ABB RAPID module: etna.mod

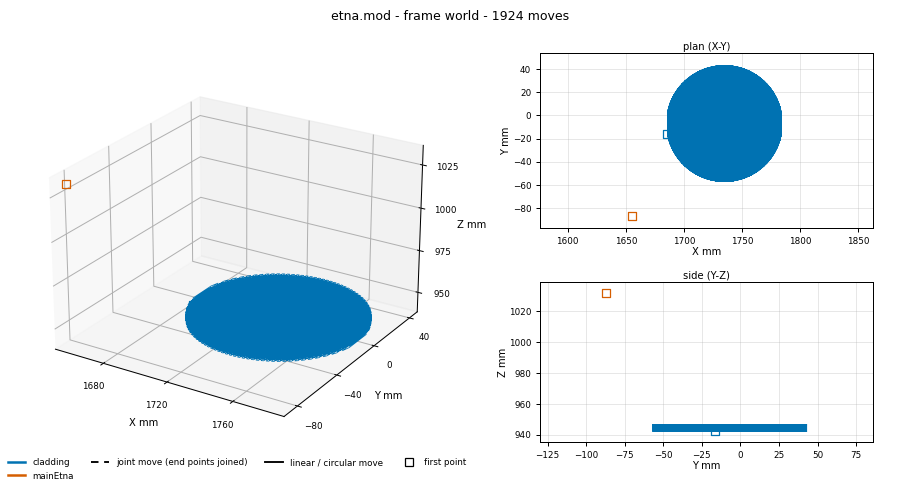
[picture p0: tool path of etna.mod in frame world, 1924 of 1924 moves have a stored position in this frame; points joined in program order, loops and branches not executed]
MODULE Etna

    PERS tooldata toolEtna:=[TRUE,[[530.0,46.8,126.6],[0.707107,0.000000,0.707107,0.000000]],[20,[70,30,123.5],[0,0,1,0],1,0,1]];
    PERS wobjdata wobjEtna:=[FALSE,TRUE,"",[[1655.0,-87.0,932.0],[1.000000,0.000000,0.000000,0.000000]],[[0,0,0],[1,0,0,0]]];

    VAR triggdata laserON;
    VAR triggdata laserOFF;

    CONST speeddata vl:=[10,500,5000,1000];


    CONST robtarget T0:=[[30.859828,70.797151,10.399975],[0.000000,0.000000,1.000000,0.000000],[0,0,-1,0],[9E+09,9E+09,9E+09,9E+09,9E+09,9E+09]];
    CONST robtarget T1:=[[30.859828,89.202857,10.399975],[0.000000,0.000000,1.000000,0.000000],[0,0,-1,0],[9E+09,9E+09,9E+09,9E+09,9E+09,9E+09]];
    CONST robtarget T2:=[[30.859828,70.797151,10.399975],[0.000000,0.000000,1.000000,0.000000],[0,0,-1,0],[9E+09,9E+09,9E+09,9E+09,9E+09,9E+09]];
    CONST robtarget T3:=[[30.859828,89.202857,10.399975],[0.000000,0.000000,1.000000,0.000000],[0,0,-1,0],[9E+09,9E+09,9E+09,9E+09,9E+09,9E+09]];
    CONST robtarget T4:=[[32.119833,94.360756,10.399975],[0.000000,0.000000,1.000000,0.000000],[0,0,-1,0],[9E+09,9E+09,9E+09,9E+09,9E+09,9E+09]];
    CONST robtarget T5:=[[32.119833,65.639251,10.399975],[0.000000,0.000000,1.000000,0.000000],[0,0,-1,0],[9E+09,9E+09,9E+09,9E+09,9E+09,9E+09]];
    CONST robtarget T6:=[[33.379837,61.953657,10.399975],[0.000000,0.000000,1.000000,0.000000],[0,0,-1,0],[9E+09,9E+09,9E+09,9E+09,9E+09,9E+09]];
    CONST robtarget T7:=[[33.379837,98.046351,10.399975],[0.000000,0.000000,1.000000,0.000000],[0,0,-1,0],[9E+09,9E+09,9E+09,9E+09,9E+09,9E+09]];
    CONST robtarget T8:=[[34.639842,101.007928,10.399975],[0.000000,0.000000,1.000000,0.000000],[0,0,-1,0],[9E+09,9E+09,9E+09,9E+09,9E+09,9E+09]];
    CONST robtarget T9:=[[34.639842,58.992080,10.399975],[0.000000,0.000000,1.000000,0.000000],[0,0,-1,0],[9E+09,9E+09,9E+09,9E+09,9E+09,9E+09]];
    CONST robtarget T10:=[[35.899846,56.444690,10.399975],[0.000000,0.000000,1.000000,0.000000],[0,0,-1,0],[9E+09,9E+09,9E+09,9E+09,9E+09,9E+09]];
    CONST robtarget T11:=[[35.899846,103.555317,10.399975],[0.000000,0.000000,1.000000,0.000000],[0,0,-1,0],[9E+09,9E+09,9E+09,9E+09,9E+09,9E+09]];
    CONST robtarget T12:=[[37.159851,105.775934,10.399975],[0.000000,0.000000,1.000000,0.000000],[0,0,-1,0],[9E+09,9E+09,9E+09,9E+09,9E+09,9E+09]];
    CONST robtarget T13:=[[37.159851,54.224074,10.399975],[0.000000,0.000000,1.000000,0.000000],[0,0,-1,0],[9E+09,9E+09,9E+09,9E+09,9E+09,9E+09]];
    CONST robtarget T14:=[[38.419855,52.240778,10.399975],[0.000000,0.000000,1.000000,0.000000],[0,0,-1,0],[9E+09,9E+09,9E+09,9E+09,9E+09,9E+09]];
    CONST robtarget T15:=[[38.419855,76.422528,10.399975],[0.000000,0.000000,1.000000,0.000000],[0,0,-1,0],[9E+09,9E+09,9E+09,9E+09,9E+09,9E+09]];
    CONST robtarget T16:=[[38.419855,83.577479,10.399975],[0.000000,0.000000,1.000000,0.000000],[0,0,-1,0],[9E+09,9E+09,9E+09,9E+09,9E+09,9E+09]];
    CONST robtarget T17:=[[38.419855,107.759230,10.399975],[0.000000,0.000000,1.000000,0.000000],[0,0,-1,0],[9E+09,9E+09,9E+09,9E+09,9E+09,9E+09]];
    CONST robtarget T18:=[[39.679860,109.560940,10.399975],[0.000000,0.000000,1.000000,0.000000],[0,0,-1,0],[9E+09,9E+09,9E+09,9E+09,9E+09,9E+09]];
    CONST robtarget T19:=[[39.679860,85.271589,10.399975],[0.000000,0.000000,1.000000,0.000000],[0,0,-1,0],[9E+09,9E+09,9E+09,9E+09,9E+09,9E+09]];
    CONST robtarget T20:=[[39.679860,74.728418,10.399975],[0.000000,0.000000,1.000000,0.000000],[0,0,-1,0],[9E+09,9E+09,9E+09,9E+09,9E+09,9E+09]];
    CONST robtarget T21:=[[39.679860,50.439068,10.399975],[0.000000,0.000000,1.000000,0.000000],[0,0,-1,0],[9E+09,9E+09,9E+09,9E+09,9E+09,9E+09]];
    CONST robtarget T22:=[[40.939864,48.787854,10.399975],[0.000000,0.000000,1.000000,0.000000],[0,0,-1,0],[9E+09,9E+09,9E+09,9E+09,9E+09,9E+09]];
    CONST robtarget T23:=[[40.939864,73.708792,10.399975],[0.000000,0.000000,1.000000,0.000000],[0,0,-1,0],[9E+09,9E+09,9E+09,9E+09,9E+09,9E+09]];
    CONST robtarget T24:=[[40.939864,86.291215,10.399975],[0.000000,0.000000,1.000000,0.000000],[0,0,-1,0],[9E+09,9E+09,9E+09,9E+09,9E+09,9E+09]];
    CONST robtarget T25:=[[40.939864,111.212154,10.399975],[0.000000,0.000000,1.000000,0.000000],[0,0,-1,0],[9E+09,9E+09,9E+09,9E+09,9E+09,9E+09]];
    CONST robtarget T26:=[[42.199869,112.721391,10.399975],[0.000000,0.000000,1.000000,0.000000],[0,0,-1,0],[9E+09,9E+09,9E+09,9E+09,9E+09,9E+09]];
    CONST robtarget T27:=[[42.199869,86.948670,10.399975],[0.000000,0.000000,1.000000,0.000000],[0,0,-1,0],[9E+09,9E+09,9E+09,9E+09,9E+09,9E+09]];
    CONST robtarget T28:=[[42.199869,73.051337,10.399975],[0.000000,0.000000,1.000000,0.000000],[0,0,-1,0],[9E+09,9E+09,9E+09,9E+09,9E+09,9E+09]];
    CONST robtarget T29:=[[42.199869,47.278617,10.399975],[0.000000,0.000000,1.000000,0.000000],[0,0,-1,0],[9E+09,9E+09,9E+09,9E+09,9E+09,9E+09]];
    CONST robtarget T30:=[[43.459873,45.884908,10.399975],[0.000000,0.000000,1.000000,0.000000],[0,0,-1,0],[9E+09,9E+09,9E+09,9E+09,9E+09,9E+09]];
    CONST robtarget T31:=[[43.459873,72.670297,10.399975],[0.000000,0.000000,1.000000,0.000000],[0,0,-1,0],[9E+09,9E+09,9E+09,9E+09,9E+09,9E+09]];
    CONST robtarget T32:=[[43.459873,87.329711,10.399975],[0.000000,0.000000,1.000000,0.000000],[0,0,-1,0],[9E+09,9E+09,9E+09,9E+09,9E+09,9E+09]];
    CONST robtarget T33:=[[43.459873,114.115099,10.399975],[0.000000,0.000000,1.000000,0.000000],[0,0,-1,0],[9E+09,9E+09,9E+09,9E+09,9E+09,9E+09]];
    CONST robtarget T34:=[[44.719878,115.412758,10.399975],[0.000000,0.000000,1.000000,0.000000],[0,0,-1,0],[9E+09,9E+09,9E+09,9E+09,9E+09,9E+09]];
    CONST robtarget T35:=[[44.719878,87.487316,10.399975],[0.000000,0.000000,1.000000,0.000000],[0,0,-1,0],[9E+09,9E+09,9E+09,9E+09,9E+09,9E+09]];
    CONST robtarget T36:=[[44.719878,72.512692,10.399975],[0.000000,0.000000,1.000000,0.000000],[0,0,-1,0],[9E+09,9E+09,9E+09,9E+09,9E+09,9E+09]];
    CONST robtarget T37:=[[44.719878,44.587250,10.399975],[0.000000,0.000000,1.000000,0.000000],[0,0,-1,0],[9E+09,9E+09,9E+09,9E+09,9E+09,9E+09]];
    CONST robtarget T38:=[[45.979882,43.373063,10.399975],[0.000000,0.000000,1.000000,0.000000],[0,0,-1,0],[9E+09,9E+09,9E+09,9E+09,9E+09,9E+09]];
    CONST robtarget T39:=[[45.979882,72.576253,10.399975],[0.000000,0.000000,1.000000,0.000000],[0,0,-1,0],[9E+09,9E+09,9E+09,9E+09,9E+09,9E+09]];
    CONST robtarget T40:=[[45.979882,87.423755,10.399975],[0.000000,0.000000,1.000000,0.000000],[0,0,-1,0],[9E+09,9E+09,9E+09,9E+09,9E+09,9E+09]];
    CONST robtarget T41:=[[45.979882,116.626944,10.399975],[0.000000,0.000000,1.000000,0.000000],[0,0,-1,0],[9E+09,9E+09,9E+09,9E+09,9E+09,9E+09]];
    CONST robtarget T42:=[[47.239887,117.767805,10.399975],[0.000000,0.000000,1.000000,0.000000],[0,0,-1,0],[9E+09,9E+09,9E+09,9E+09,9E+09,9E+09]];
    CONST robtarget T43:=[[47.239887,87.152583,10.399975],[0.000000,0.000000,1.000000,0.000000],[0,0,-1,0],[9E+09,9E+09,9E+09,9E+09,9E+09,9E+09]];
    CONST robtarget T44:=[[47.239887,72.847425,10.399975],[0.000000,0.000000,1.000000,0.000000],[0,0,-1,0],[9E+09,9E+09,9E+09,9E+09,9E+09,9E+09]];
    CONST robtarget T45:=[[47.239887,42.232203,10.399975],[0.000000,0.000000,1.000000,0.000000],[0,0,-1,0],[9E+09,9E+09,9E+09,9E+09,9E+09,9E+09]];
    CONST robtarget T46:=[[48.499891,41.180273,10.399975],[0.000000,0.000000,1.000000,0.000000],[0,0,-1,0],[9E+09,9E+09,9E+09,9E+09,9E+09,9E+09]];
    CONST robtarget T47:=[[48.499891,73.379202,10.399975],[0.000000,0.000000,1.000000,0.000000],[0,0,-1,0],[9E+09,9E+09,9E+09,9E+09,9E+09,9E+09]];
    CONST robtarget T48:=[[48.499891,86.620805,10.399975],[0.000000,0.000000,1.000000,0.000000],[0,0,-1,0],[9E+09,9E+09,9E+09,9E+09,9E+09,9E+09]];
    CONST robtarget T49:=[[48.499891,118.819735,10.399975],[0.000000,0.000000,1.000000,0.000000],[0,0,-1,0],[9E+09,9E+09,9E+09,9E+09,9E+09,9E+09]];
    CONST robtarget T50:=[[49.759896,119.803025,10.399975],[0.000000,0.000000,1.000000,0.000000],[0,0,-1,0],[9E+09,9E+09,9E+09,9E+09,9E+09,9E+09]];
    CONST robtarget T51:=[[49.759896,85.779969,10.399975],[0.000000,0.000000,1.000000,0.000000],[0,0,-1,0],[9E+09,9E+09,9E+09,9E+09,9E+09,9E+09]];
    CONST robtarget T52:=[[49.759896,74.220038,10.399975],[0.000000,0.000000,1.000000,0.000000],[0,0,-1,0],[9E+09,9E+09,9E+09,9E+09,9E+09,9E+09]];
    CONST robtarget T53:=[[49.759896,40.196983,10.399975],[0.000000,0.000000,1.000000,0.000000],[0,0,-1,0],[9E+09,9E+09,9E+09,9E+09,9E+09,9E+09]];
    CONST robtarget T54:=[[51.019900,39.265681,10.399975],[0.000000,0.000000,1.000000,0.000000],[0,0,-1,0],[9E+09,9E+09,9E+09,9E+09,9E+09,9E+09]];
    CONST robtarget T55:=[[51.019900,75.547902,10.399975],[0.000000,0.000000,1.000000,0.000000],[0,0,-1,0],[9E+09,9E+09,9E+09,9E+09,9E+09,9E+09]];
    CONST robtarget T56:=[[51.019900,84.452106,10.399975],[0.000000,0.000000,1.000000,0.000000],[0,0,-1,0],[9E+09,9E+09,9E+09,9E+09,9E+09,9E+09]];
    CONST robtarget T57:=[[51.019900,120.734326,10.399975],[0.000000,0.000000,1.000000,0.000000],[0,0,-1,0],[9E+09,9E+09,9E+09,9E+09,9E+09,9E+09]];
    CONST robtarget T58:=[[52.279905,121.607260,10.399975],[0.000000,0.000000,1.000000,0.000000],[0,0,-1,0],[9E+09,9E+09,9E+09,9E+09,9E+09,9E+09]];
    CONST robtarget T59:=[[52.279905,81.789524,10.399975],[0.000000,0.000000,1.000000,0.000000],[0,0,-1,0],[9E+09,9E+09,9E+09,9E+09,9E+09,9E+09]];
    CONST robtarget T60:=[[52.279905,78.210483,10.399975],[0.000000,0.000000,1.000000,0.000000],[0,0,-1,0],[9E+09,9E+09,9E+09,9E+09,9E+09,9E+09]];
    CONST robtarget T61:=[[52.279905,38.392748,10.399975],[0.000000,0.000000,1.000000,0.000000],[0,0,-1,0],[9E+09,9E+09,9E+09,9E+09,9E+09,9E+09]];
    CONST robtarget T62:=[[53.539909,37.589739,10.399975],[0.000000,0.000000,1.000000,0.000000],[0,0,-1,0],[9E+09,9E+09,9E+09,9E+09,9E+09,9E+09]];
    CONST robtarget T63:=[[53.539909,122.410268,10.399975],[0.000000,0.000000,1.000000,0.000000],[0,0,-1,0],[9E+09,9E+09,9E+09,9E+09,9E+09,9E+09]];
    CONST robtarget T64:=[[54.799914,123.174878,10.399975],[0.000000,0.000000,1.000000,0.000000],[0,0,-1,0],[9E+09,9E+09,9E+09,9E+09,9E+09,9E+09]];
    CONST robtarget T65:=[[54.799914,36.825129,10.399975],[0.000000,0.000000,1.000000,0.000000],[0,0,-1,0],[9E+09,9E+09,9E+09,9E+09,9E+09,9E+09]];
    CONST robtarget T66:=[[56.059918,36.110177,10.399975],[0.000000,0.000000,1.000000,0.000000],[0,0,-1,0],[9E+09,9E+09,9E+09,9E+09,9E+09,9E+09]];
    CONST robtarget T67:=[[56.059918,123.889831,10.399975],[0.000000,0.000000,1.000000,0.000000],[0,0,-1,0],[9E+09,9E+09,9E+09,9E+09,9E+09,9E+09]];
    CONST robtarget T68:=[[57.319923,124.546114,10.399975],[0.000000,0.000000,1.000000,0.000000],[0,0,-1,0],[9E+09,9E+09,9E+09,9E+09,9E+09,9E+09]];
    CONST robtarget T69:=[[57.319923,35.453894,10.399975],[0.000000,0.000000,1.000000,0.000000],[0,0,-1,0],[9E+09,9E+09,9E+09,9E+09,9E+09,9E+09]];
    CONST robtarget T70:=[[58.579927,34.827050,10.399975],[0.000000,0.000000,1.000000,0.000000],[0,0,-1,0],[9E+09,9E+09,9E+09,9E+09,9E+09,9E+09]];
    CONST robtarget T71:=[[58.579927,125.172958,10.399975],[0.000000,0.000000,1.000000,0.000000],[0,0,-1,0],[9E+09,9E+09,9E+09,9E+09,9E+09,9E+09]];
    CONST robtarget T72:=[[59.839932,125.745278,10.399975],[0.000000,0.000000,1.000000,0.000000],[0,0,-1,0],[9E+09,9E+09,9E+09,9E+09,9E+09,9E+09]];
    CONST robtarget T73:=[[59.839932,34.254730,10.399975],[0.000000,0.000000,1.000000,0.000000],[0,0,-1,0],[9E+09,9E+09,9E+09,9E+09,9E+09,9E+09]];
    CONST robtarget T74:=[[61.099936,33.722290,10.399975],[0.000000,0.000000,1.000000,0.000000],[0,0,-1,0],[9E+09,9E+09,9E+09,9E+09,9E+09,9E+09]];
    CONST robtarget T75:=[[61.099936,126.277717,10.399975],[0.000000,0.000000,1.000000,0.000000],[0,0,-1,0],[9E+09,9E+09,9E+09,9E+09,9E+09,9E+09]];
    CONST robtarget T76:=[[62.359941,126.783143,10.399975],[0.000000,0.000000,1.000000,0.000000],[0,0,-1,0],[9E+09,9E+09,9E+09,9E+09,9E+09,9E+09]];
    CONST robtarget T77:=[[62.359941,33.216864,10.399975],[0.000000,0.000000,1.000000,0.000000],[0,0,-1,0],[9E+09,9E+09,9E+09,9E+09,9E+09,9E+09]];
    CONST robtarget T78:=[[63.619945,32.772318,10.399975],[0.000000,0.000000,1.000000,0.000000],[0,0,-1,0],[9E+09,9E+09,9E+09,9E+09,9E+09,9E+09]];
    CONST robtarget T79:=[[63.619945,127.227690,10.399975],[0.000000,0.000000,1.000000,0.000000],[0,0,-1,0],[9E+09,9E+09,9E+09,9E+09,9E+09,9E+09]];
    CONST robtarget T80:=[[64.879950,127.652167,10.399975],[0.000000,0.000000,1.000000,0.000000],[0,0,-1,0],[9E+09,9E+09,9E+09,9E+09,9E+09,9E+09]];
    CONST robtarget T81:=[[64.879950,32.347841,10.399975],[0.000000,0.000000,1.000000,0.000000],[0,0,-1,0],[9E+09,9E+09,9E+09,9E+09,9E+09,9E+09]];
    CONST robtarget T82:=[[66.139954,31.969479,10.399975],[0.000000,0.000000,1.000000,0.000000],[0,0,-1,0],[9E+09,9E+09,9E+09,9E+09,9E+09,9E+09]];
    CONST robtarget T83:=[[66.139954,128.030529,10.399975],[0.000000,0.000000,1.000000,0.000000],[0,0,-1,0],[9E+09,9E+09,9E+09,9E+09,9E+09,9E+09]];
    CONST robtarget T84:=[[67.399959,128.374988,10.399975],[0.000000,0.000000,1.000000,0.000000],[0,0,-1,0],[9E+09,9E+09,9E+09,9E+09,9E+09,9E+09]];
    CONST robtarget T85:=[[67.399959,31.625019,10.399975],[0.000000,0.000000,1.000000,0.000000],[0,0,-1,0],[9E+09,9E+09,9E+09,9E+09,9E+09,9E+09]];
    CONST robtarget T86:=[[68.659963,31.307526,10.399975],[0.000000,0.000000,1.000000,0.000000],[0,0,-1,0],[9E+09,9E+09,9E+09,9E+09,9E+09,9E+09]];
    CONST robtarget T87:=[[68.659963,128.692481,10.399975],[0.000000,0.000000,1.000000,0.000000],[0,0,-1,0],[9E+09,9E+09,9E+09,9E+09,9E+09,9E+09]];
    CONST robtarget T88:=[[69.919968,128.960575,10.399975],[0.000000,0.000000,1.000000,0.000000],[0,0,-1,0],[9E+09,9E+09,9E+09,9E+09,9E+09,9E+09]];
    CONST robtarget T89:=[[69.919968,31.039433,10.399975],[0.000000,0.000000,1.000000,0.000000],[0,0,-1,0],[9E+09,9E+09,9E+09,9E+09,9E+09,9E+09]];
    CONST robtarget T90:=[[71.179972,30.786444,10.399975],[0.000000,0.000000,1.000000,0.000000],[0,0,-1,0],[9E+09,9E+09,9E+09,9E+09,9E+09,9E+09]];
    CONST robtarget T91:=[[71.179972,129.213563,10.399975],[0.000000,0.000000,1.000000,0.000000],[0,0,-1,0],[9E+09,9E+09,9E+09,9E+09,9E+09,9E+09]];
    CONST robtarget T92:=[[72.439977,129.413129,10.399975],[0.000000,0.000000,1.000000,0.000000],[0,0,-1,0],[9E+09,9E+09,9E+09,9E+09,9E+09,9E+09]];
    CONST robtarget T93:=[[72.439977,30.586879,10.399975],[0.000000,0.000000,1.000000,0.000000],[0,0,-1,0],[9E+09,9E+09,9E+09,9E+09,9E+09,9E+09]];
    CONST robtarget T94:=[[73.699981,30.406130,10.399975],[0.000000,0.000000,1.000000,0.000000],[0,0,-1,0],[9E+09,9E+09,9E+09,9E+09,9E+09,9E+09]];
    CONST robtarget T95:=[[73.699981,40.937335,10.399975],[0.000000,0.000000,1.000000,0.000000],[0,0,-1,0],[9E+09,9E+09,9E+09,9E+09,9E+09,9E+09]];
    CONST robtarget T96:=[[73.699981,49.062665,10.399975],[0.000000,0.000000,1.000000,0.000000],[0,0,-1,0],[9E+09,9E+09,9E+09,9E+09,9E+09,9E+09]];
    CONST robtarget T97:=[[73.699981,75.937339,10.399975],[0.000000,0.000000,1.000000,0.000000],[0,0,-1,0],[9E+09,9E+09,9E+09,9E+09,9E+09,9E+09]];
    CONST robtarget T98:=[[73.699981,84.062668,10.399975],[0.000000,0.000000,1.000000,0.000000],[0,0,-1,0],[9E+09,9E+09,9E+09,9E+09,9E+09,9E+09]];
    CONST robtarget T99:=[[73.699981,110.937342,10.399975],[0.000000,0.000000,1.000000,0.000000],[0,0,-1,0],[9E+09,9E+09,9E+09,9E+09,9E+09,9E+09]];
    CONST robtarget T100:=[[73.699981,119.062672,10.399975],[0.000000,0.000000,1.000000,0.000000],[0,0,-1,0],[9E+09,9E+09,9E+09,9E+09,9E+09,9E+09]];
    CONST robtarget T101:=[[73.699981,129.593877,10.399975],[0.000000,0.000000,1.000000,0.000000],[0,0,-1,0],[9E+09,9E+09,9E+09,9E+09,9E+09,9E+09]];
    CONST robtarget T102:=[[74.959986,129.735844,10.399975],[0.000000,0.000000,1.000000,0.000000],[0,0,-1,0],[9E+09,9E+09,9E+09,9E+09,9E+09,9E+09]];
    CONST robtarget T103:=[[74.959986,120.544921,10.399975],[0.000000,0.000000,1.000000,0.000000],[0,0,-1,0],[9E+09,9E+09,9E+09,9E+09,9E+09,9E+09]];
    CONST robtarget T104:=[[74.959986,109.455091,10.399975],[0.000000,0.000000,1.000000,0.000000],[0,0,-1,0],[9E+09,9E+09,9E+09,9E+09,9E+09,9E+09]];
    CONST robtarget T105:=[[74.959986,85.544918,10.399975],[0.000000,0.000000,1.000000,0.000000],[0,0,-1,0],[9E+09,9E+09,9E+09,9E+09,9E+09,9E+09]];
    CONST robtarget T106:=[[74.959986,74.455090,10.399975],[0.000000,0.000000,1.000000,0.000000],[0,0,-1,0],[9E+09,9E+09,9E+09,9E+09,9E+09,9E+09]];
    CONST robtarget T107:=[[74.959986,50.544916,10.399975],[0.000000,0.000000,1.000000,0.000000],[0,0,-1,0],[9E+09,9E+09,9E+09,9E+09,9E+09,9E+09]];
    CONST robtarget T108:=[[74.959986,39.455086,10.399975],[0.000000,0.000000,1.000000,0.000000],[0,0,-1,0],[9E+09,9E+09,9E+09,9E+09,9E+09,9E+09]];
    CONST robtarget T109:=[[74.959986,30.264163,10.399975],[0.000000,0.000000,1.000000,0.000000],[0,0,-1,0],[9E+09,9E+09,9E+09,9E+09,9E+09,9E+09]];
    CONST robtarget T110:=[[76.219990,30.153959,10.399975],[0.000000,0.000000,1.000000,0.000000],[0,0,-1,0],[9E+09,9E+09,9E+09,9E+09,9E+09,9E+09]];
    CONST robtarget T111:=[[76.219990,38.524551,10.399975],[0.000000,0.000000,1.000000,0.000000],[0,0,-1,0],[9E+09,9E+09,9E+09,9E+09,9E+09,9E+09]];
    CONST robtarget T112:=[[76.219990,51.475451,10.399975],[0.000000,0.000000,1.000000,0.000000],[0,0,-1,0],[9E+09,9E+09,9E+09,9E+09,9E+09,9E+09]];
    CONST robtarget T113:=[[76.219990,73.524553,10.399975],[0.000000,0.000000,1.000000,0.000000],[0,0,-1,0],[9E+09,9E+09,9E+09,9E+09,9E+09,9E+09]];
    CONST robtarget T114:=[[76.219990,86.475455,10.399975],[0.000000,0.000000,1.000000,0.000000],[0,0,-1,0],[9E+09,9E+09,9E+09,9E+09,9E+09,9E+09]];
    CONST robtarget T115:=[[76.219990,108.524556,10.399975],[0.000000,0.000000,1.000000,0.000000],[0,0,-1,0],[9E+09,9E+09,9E+09,9E+09,9E+09,9E+09]];
    CONST robtarget T116:=[[76.219990,121.475457,10.399975],[0.000000,0.000000,1.000000,0.000000],[0,0,-1,0],[9E+09,9E+09,9E+09,9E+09,9E+09,9E+09]];
    CONST robtarget T117:=[[76.219990,129.846049,10.399975],[0.000000,0.000000,1.000000,0.000000],[0,0,-1,0],[9E+09,9E+09,9E+09,9E+09,9E+09,9E+09]];
    CONST robtarget T118:=[[77.479995,129.931001,10.399975],[0.000000,0.000000,1.000000,0.000000],[0,0,-1,0],[9E+09,9E+09,9E+09,9E+09,9E+09,9E+09]];
    CONST robtarget T119:=[[77.479995,122.050628,10.399975],[0.000000,0.000000,1.000000,0.000000],[0,0,-1,0],[9E+09,9E+09,9E+09,9E+09,9E+09,9E+09]];
    CONST robtarget T120:=[[77.479995,107.949384,10.399975],[0.000000,0.000000,1.000000,0.000000],[0,0,-1,0],[9E+09,9E+09,9E+09,9E+09,9E+09,9E+09]];
    CONST robtarget T121:=[[77.479995,87.050626,10.399975],[0.000000,0.000000,1.000000,0.000000],[0,0,-1,0],[9E+09,9E+09,9E+09,9E+09,9E+09,9E+09]];
    CONST robtarget T122:=[[77.479995,72.949381,10.399975],[0.000000,0.000000,1.000000,0.000000],[0,0,-1,0],[9E+09,9E+09,9E+09,9E+09,9E+09,9E+09]];
    CONST robtarget T123:=[[77.479995,52.050624,10.399975],[0.000000,0.000000,1.000000,0.000000],[0,0,-1,0],[9E+09,9E+09,9E+09,9E+09,9E+09,9E+09]];
    CONST robtarget T124:=[[77.479995,37.949379,10.399975],[0.000000,0.000000,1.000000,0.000000],[0,0,-1,0],[9E+09,9E+09,9E+09,9E+09,9E+09,9E+09]];
    CONST robtarget T125:=[[77.479995,30.069007,10.399975],[0.000000,0.000000,1.000000,0.000000],[0,0,-1,0],[9E+09,9E+09,9E+09,9E+09,9E+09,9E+09]];
    CONST robtarget T126:=[[78.739999,30.028279,10.399975],[0.000000,0.000000,1.000000,0.000000],[0,0,-1,0],[9E+09,9E+09,9E+09,9E+09,9E+09,9E+09]];
    CONST robtarget T127:=[[78.739999,37.608991,10.399975],[0.000000,0.000000,1.000000,0.000000],[0,0,-1,0],[9E+09,9E+09,9E+09,9E+09,9E+09,9E+09]];
    CONST robtarget T128:=[[78.739999,52.391011,10.399975],[0.000000,0.000000,1.000000,0.000000],[0,0,-1,0],[9E+09,9E+09,9E+09,9E+09,9E+09,9E+09]];
    CONST robtarget T129:=[[78.739999,72.608994,10.399975],[0.000000,0.000000,1.000000,0.000000],[0,0,-1,0],[9E+09,9E+09,9E+09,9E+09,9E+09,9E+09]];
    CONST robtarget T130:=[[78.739999,87.391014,10.399975],[0.000000,0.000000,1.000000,0.000000],[0,0,-1,0],[9E+09,9E+09,9E+09,9E+09,9E+09,9E+09]];
    CONST robtarget T131:=[[78.739999,107.608996,10.399975],[0.000000,0.000000,1.000000,0.000000],[0,0,-1,0],[9E+09,9E+09,9E+09,9E+09,9E+09,9E+09]];
    CONST robtarget T132:=[[78.739999,122.391017,10.399975],[0.000000,0.000000,1.000000,0.000000],[0,0,-1,0],[9E+09,9E+09,9E+09,9E+09,9E+09,9E+09]];
    CONST robtarget T133:=[[78.739999,129.971729,10.399975],[0.000000,0.000000,1.000000,0.000000],[0,0,-1,0],[9E+09,9E+09,9E+09,9E+09,9E+09,9E+09]];
    CONST robtarget T134:=[[80.000004,130.000008,10.399975],[0.000000,0.000000,1.000000,0.000000],[0,0,-1,0],[9E+09,9E+09,9E+09,9E+09,9E+09,9E+09]];
    CONST robtarget T135:=[[80.000004,122.487319,10.399975],[0.000000,0.000000,1.000000,0.000000],[0,0,-1,0],[9E+09,9E+09,9E+09,9E+09,9E+09,9E+09]];
    CONST robtarget T136:=[[80.000004,107.512696,10.399975],[0.000000,0.000000,1.000000,0.000000],[0,0,-1,0],[9E+09,9E+09,9E+09,9E+09,9E+09,9E+09]];
    CONST robtarget T137:=[[80.000004,87.487316,10.399975],[0.000000,0.000000,1.000000,0.000000],[0,0,-1,0],[9E+09,9E+09,9E+09,9E+09,9E+09,9E+09]];
    CONST robtarget T138:=[[80.000004,72.512692,10.399975],[0.000000,0.000000,1.000000,0.000000],[0,0,-1,0],[9E+09,9E+09,9E+09,9E+09,9E+09,9E+09]];
    CONST robtarget T139:=[[80.000004,52.487312,10.399975],[0.000000,0.000000,1.000000,0.000000],[0,0,-1,0],[9E+09,9E+09,9E+09,9E+09,9E+09,9E+09]];
    CONST robtarget T140:=[[80.000004,37.512688,10.399975],[0.000000,0.000000,1.000000,0.000000],[0,0,-1,0],[9E+09,9E+09,9E+09,9E+09,9E+09,9E+09]];
    CONST robtarget T141:=[[80.000004,30.000000,10.399975],[0.000000,0.000000,1.000000,0.000000],[0,0,-1,0],[9E+09,9E+09,9E+09,9E+09,9E+09,9E+09]];
    CONST robtarget T142:=[[81.260008,30.028279,10.399975],[0.000000,0.000000,1.000000,0.000000],[0,0,-1,0],[9E+09,9E+09,9E+09,9E+09,9E+09,9E+09]];
    CONST robtarget T143:=[[81.260008,37.608991,10.399975],[0.000000,0.000000,1.000000,0.000000],[0,0,-1,0],[9E+09,9E+09,9E+09,9E+09,9E+09,9E+09]];
    CONST robtarget T144:=[[81.260008,52.391011,10.399975],[0.000000,0.000000,1.000000,0.000000],[0,0,-1,0],[9E+09,9E+09,9E+09,9E+09,9E+09,9E+09]];
    CONST robtarget T145:=[[81.260008,72.608994,10.399975],[0.000000,0.000000,1.000000,0.000000],[0,0,-1,0],[9E+09,9E+09,9E+09,9E+09,9E+09,9E+09]];
    CONST robtarget T146:=[[81.260008,87.391014,10.399975],[0.000000,0.000000,1.000000,0.000000],[0,0,-1,0],[9E+09,9E+09,9E+09,9E+09,9E+09,9E+09]];
    CONST robtarget T147:=[[81.260008,107.608996,10.399975],[0.000000,0.000000,1.000000,0.000000],[0,0,-1,0],[9E+09,9E+09,9E+09,9E+09,9E+09,9E+09]];
    CONST robtarget T148:=[[81.260008,122.391017,10.399975],[0.000000,0.000000,1.000000,0.000000],[0,0,-1,0],[9E+09,9E+09,9E+09,9E+09,9E+09,9E+09]];
    CONST robtarget T149:=[[81.260008,129.971729,10.399975],[0.000000,0.000000,1.000000,0.000000],[0,0,-1,0],[9E+09,9E+09,9E+09,9E+09,9E+09,9E+09]];
    CONST robtarget T150:=[[82.520013,129.931001,10.399975],[0.000000,0.000000,1.000000,0.000000],[0,0,-1,0],[9E+09,9E+09,9E+09,9E+09,9E+09,9E+09]];
    CONST robtarget T151:=[[82.520013,122.050628,10.399975],[0.000000,0.000000,1.000000,0.000000],[0,0,-1,0],[9E+09,9E+09,9E+09,9E+09,9E+09,9E+09]];
    CONST robtarget T152:=[[82.520013,107.949384,10.399975],[0.000000,0.000000,1.000000,0.000000],[0,0,-1,0],[9E+09,9E+09,9E+09,9E+09,9E+09,9E+09]];
    CONST robtarget T153:=[[82.520013,87.050626,10.399975],[0.000000,0.000000,1.000000,0.000000],[0,0,-1,0],[9E+09,9E+09,9E+09,9E+09,9E+09,9E+09]];
    CONST robtarget T154:=[[82.520013,72.949381,10.399975],[0.000000,0.000000,1.000000,0.000000],[0,0,-1,0],[9E+09,9E+09,9E+09,9E+09,9E+09,9E+09]];
    CONST robtarget T155:=[[82.520013,52.050624,10.399975],[0.000000,0.000000,1.000000,0.000000],[0,0,-1,0],[9E+09,9E+09,9E+09,9E+09,9E+09,9E+09]];
    CONST robtarget T156:=[[82.520013,37.949379,10.399975],[0.000000,0.000000,1.000000,0.000000],[0,0,-1,0],[9E+09,9E+09,9E+09,9E+09,9E+09,9E+09]];
    CONST robtarget T157:=[[82.520013,30.069007,10.399975],[0.000000,0.000000,1.000000,0.000000],[0,0,-1,0],[9E+09,9E+09,9E+09,9E+09,9E+09,9E+09]];
    CONST robtarget T158:=[[83.780017,30.153959,10.399975],[0.000000,0.000000,1.000000,0.000000],[0,0,-1,0],[9E+09,9E+09,9E+09,9E+09,9E+09,9E+09]];
    CONST robtarget T159:=[[83.780017,38.524551,10.399975],[0.000000,0.000000,1.000000,0.000000],[0,0,-1,0],[9E+09,9E+09,9E+09,9E+09,9E+09,9E+09]];
    CONST robtarget T160:=[[83.780017,51.475451,10.399975],[0.000000,0.000000,1.000000,0.000000],[0,0,-1,0],[9E+09,9E+09,9E+09,9E+09,9E+09,9E+09]];
    CONST robtarget T161:=[[83.780017,73.524553,10.399975],[0.000000,0.000000,1.000000,0.000000],[0,0,-1,0],[9E+09,9E+09,9E+09,9E+09,9E+09,9E+09]];
    CONST robtarget T162:=[[83.780017,86.475455,10.399975],[0.000000,0.000000,1.000000,0.000000],[0,0,-1,0],[9E+09,9E+09,9E+09,9E+09,9E+09,9E+09]];
    CONST robtarget T163:=[[83.780017,108.524556,10.399975],[0.000000,0.000000,1.000000,0.000000],[0,0,-1,0],[9E+09,9E+09,9E+09,9E+09,9E+09,9E+09]];
    CONST robtarget T164:=[[83.780017,121.475457,10.399975],[0.000000,0.000000,1.000000,0.000000],[0,0,-1,0],[9E+09,9E+09,9E+09,9E+09,9E+09,9E+09]];
    CONST robtarget T165:=[[83.780017,129.846049,10.399975],[0.000000,0.000000,1.000000,0.000000],[0,0,-1,0],[9E+09,9E+09,9E+09,9E+09,9E+09,9E+09]];
    CONST robtarget T166:=[[85.040022,129.735844,10.399975],[0.000000,0.000000,1.000000,0.000000],[0,0,-1,0],[9E+09,9E+09,9E+09,9E+09,9E+09,9E+09]];
    CONST robtarget T167:=[[85.040022,120.544921,10.399975],[0.000000,0.000000,1.000000,0.000000],[0,0,-1,0],[9E+09,9E+09,9E+09,9E+09,9E+09,9E+09]];
    CONST robtarget T168:=[[85.040022,109.455091,10.399975],[0.000000,0.000000,1.000000,0.000000],[0,0,-1,0],[9E+09,9E+09,9E+09,9E+09,9E+09,9E+09]];
    CONST robtarget T169:=[[85.040022,85.544918,10.399975],[0.000000,0.000000,1.000000,0.000000],[0,0,-1,0],[9E+09,9E+09,9E+09,9E+09,9E+09,9E+09]];
    CONST robtarget T170:=[[85.040022,74.455090,10.399975],[0.000000,0.000000,1.000000,0.000000],[0,0,-1,0],[9E+09,9E+09,9E+09,9E+09,9E+09,9E+09]];
    CONST robtarget T171:=[[85.040022,50.544916,10.399975],[0.000000,0.000000,1.000000,0.000000],[0,0,-1,0],[9E+09,9E+09,9E+09,9E+09,9E+09,9E+09]];
    CONST robtarget T172:=[[85.040022,39.455086,10.399975],[0.000000,0.000000,1.000000,0.000000],[0,0,-1,0],[9E+09,9E+09,9E+09,9E+09,9E+09,9E+09]];
    CONST robtarget T173:=[[85.040022,30.264163,10.399975],[0.000000,0.000000,1.000000,0.000000],[0,0,-1,0],[9E+09,9E+09,9E+09,9E+09,9E+09,9E+09]];
    CONST robtarget T174:=[[86.300026,30.406130,10.399975],[0.000000,0.000000,1.000000,0.000000],[0,0,-1,0],[9E+09,9E+09,9E+09,9E+09,9E+09,9E+09]];
    CONST robtarget T175:=[[86.300026,40.937335,10.399975],[0.000000,0.000000,1.000000,0.000000],[0,0,-1,0],[9E+09,9E+09,9E+09,9E+09,9E+09,9E+09]];
    CONST robtarget T176:=[[86.300026,49.062665,10.399975],[0.000000,0.000000,1.000000,0.000000],[0,0,-1,0],[9E+09,9E+09,9E+09,9E+09,9E+09,9E+09]];
    CONST robtarget T177:=[[86.300026,75.937339,10.399975],[0.000000,0.000000,1.000000,0.000000],[0,0,-1,0],[9E+09,9E+09,9E+09,9E+09,9E+09,9E+09]];
    CONST robtarget T178:=[[86.300026,84.062668,10.399975],[0.000000,0.000000,1.000000,0.000000],[0,0,-1,0],[9E+09,9E+09,9E+09,9E+09,9E+09,9E+09]];
    CONST robtarget T179:=[[86.300026,110.937342,10.399975],[0.000000,0.000000,1.000000,0.000000],[0,0,-1,0],[9E+09,9E+09,9E+09,9E+09,9E+09,9E+09]];
    CONST robtarget T180:=[[86.300026,119.062672,10.399975],[0.000000,0.000000,1.000000,0.000000],[0,0,-1,0],[9E+09,9E+09,9E+09,9E+09,9E+09,9E+09]];
    CONST robtarget T181:=[[86.300026,129.593877,10.399975],[0.000000,0.000000,1.000000,0.000000],[0,0,-1,0],[9E+09,9E+09,9E+09,9E+09,9E+09,9E+09]];
    CONST robtarget T182:=[[87.560031,129.413129,10.399975],[0.000000,0.000000,1.000000,0.000000],[0,0,-1,0],[9E+09,9E+09,9E+09,9E+09,9E+09,9E+09]];
    CONST robtarget T183:=[[87.560031,30.586879,10.399975],[0.000000,0.000000,1.000000,0.000000],[0,0,-1,0],[9E+09,9E+09,9E+09,9E+09,9E+09,9E+09]];
    CONST robtarget T184:=[[88.820035,30.786444,10.399975],[0.000000,0.000000,1.000000,0.000000],[0,0,-1,0],[9E+09,9E+09,9E+09,9E+09,9E+09,9E+09]];
    CONST robtarget T185:=[[88.820035,129.213563,10.399975],[0.000000,0.000000,1.000000,0.000000],[0,0,-1,0],[9E+09,9E+09,9E+09,9E+09,9E+09,9E+09]];
    CONST robtarget T186:=[[90.080040,128.960575,10.399975],[0.000000,0.000000,1.000000,0.000000],[0,0,-1,0],[9E+09,9E+09,9E+09,9E+09,9E+09,9E+09]];
    CONST robtarget T187:=[[90.080040,31.039433,10.399975],[0.000000,0.000000,1.000000,0.000000],[0,0,-1,0],[9E+09,9E+09,9E+09,9E+09,9E+09,9E+09]];
    CONST robtarget T188:=[[91.340044,31.307526,10.399975],[0.000000,0.000000,1.000000,0.000000],[0,0,-1,0],[9E+09,9E+09,9E+09,9E+09,9E+09,9E+09]];
    CONST robtarget T189:=[[91.340044,128.692481,10.399975],[0.000000,0.000000,1.000000,0.000000],[0,0,-1,0],[9E+09,9E+09,9E+09,9E+09,9E+09,9E+09]];
    CONST robtarget T190:=[[92.600049,128.374988,10.399975],[0.000000,0.000000,1.000000,0.000000],[0,0,-1,0],[9E+09,9E+09,9E+09,9E+09,9E+09,9E+09]];
    CONST robtarget T191:=[[92.600049,31.625019,10.399975],[0.000000,0.000000,1.000000,0.000000],[0,0,-1,0],[9E+09,9E+09,9E+09,9E+09,9E+09,9E+09]];
    CONST robtarget T192:=[[93.860053,31.969479,10.399975],[0.000000,0.000000,1.000000,0.000000],[0,0,-1,0],[9E+09,9E+09,9E+09,9E+09,9E+09,9E+09]];
    CONST robtarget T193:=[[93.860053,128.030529,10.399975],[0.000000,0.000000,1.000000,0.000000],[0,0,-1,0],[9E+09,9E+09,9E+09,9E+09,9E+09,9E+09]];
    CONST robtarget T194:=[[95.120058,127.652167,10.399975],[0.000000,0.000000,1.000000,0.000000],[0,0,-1,0],[9E+09,9E+09,9E+09,9E+09,9E+09,9E+09]];
    CONST robtarget T195:=[[95.120058,32.347841,10.399975],[0.000000,0.000000,1.000000,0.000000],[0,0,-1,0],[9E+09,9E+09,9E+09,9E+09,9E+09,9E+09]];
    CONST robtarget T196:=[[96.380062,32.772318,10.399975],[0.000000,0.000000,1.000000,0.000000],[0,0,-1,0],[9E+09,9E+09,9E+09,9E+09,9E+09,9E+09]];
    CONST robtarget T197:=[[96.380062,127.227690,10.399975],[0.000000,0.000000,1.000000,0.000000],[0,0,-1,0],[9E+09,9E+09,9E+09,9E+09,9E+09,9E+09]];
    CONST robtarget T198:=[[97.640067,126.783143,10.399975],[0.000000,0.000000,1.000000,0.000000],[0,0,-1,0],[9E+09,9E+09,9E+09,9E+09,9E+09,9E+09]];
    CONST robtarget T199:=[[97.640067,33.216864,10.399975],[0.000000,0.000000,1.000000,0.000000],[0,0,-1,0],[9E+09,9E+09,9E+09,9E+09,9E+09,9E+09]];
    CONST robtarget T200:=[[98.900071,33.722290,10.399975],[0.000000,0.000000,1.000000,0.000000],[0,0,-1,0],[9E+09,9E+09,9E+09,9E+09,9E+09,9E+09]];
    CONST robtarget T201:=[[98.900071,126.277717,10.399975],[0.000000,0.000000,1.000000,0.000000],[0,0,-1,0],[9E+09,9E+09,9E+09,9E+09,9E+09,9E+09]];
    CONST robtarget T202:=[[100.160076,125.745278,10.399975],[0.000000,0.000000,1.000000,0.000000],[0,0,-1,0],[9E+09,9E+09,9E+09,9E+09,9E+09,9E+09]];
    CONST robtarget T203:=[[100.160076,34.254730,10.399975],[0.000000,0.000000,1.000000,0.000000],[0,0,-1,0],[9E+09,9E+09,9E+09,9E+09,9E+09,9E+09]];
    CONST robtarget T204:=[[101.420080,34.827050,10.399975],[0.000000,0.000000,1.000000,0.000000],[0,0,-1,0],[9E+09,9E+09,9E+09,9E+09,9E+09,9E+09]];
    CONST robtarget T205:=[[101.420080,125.172958,10.399975],[0.000000,0.000000,1.000000,0.000000],[0,0,-1,0],[9E+09,9E+09,9E+09,9E+09,9E+09,9E+09]];
    CONST robtarget T206:=[[102.680085,124.546114,10.399975],[0.000000,0.000000,1.000000,0.000000],[0,0,-1,0],[9E+09,9E+09,9E+09,9E+09,9E+09,9E+09]];
    CONST robtarget T207:=[[102.680085,35.453894,10.399975],[0.000000,0.000000,1.000000,0.000000],[0,0,-1,0],[9E+09,9E+09,9E+09,9E+09,9E+09,9E+09]];
    CONST robtarget T208:=[[103.940089,36.110177,10.399975],[0.000000,0.000000,1.000000,0.000000],[0,0,-1,0],[9E+09,9E+09,9E+09,9E+09,9E+09,9E+09]];
    CONST robtarget T209:=[[103.940089,123.889831,10.399975],[0.000000,0.000000,1.000000,0.000000],[0,0,-1,0],[9E+09,9E+09,9E+09,9E+09,9E+09,9E+09]];
    CONST robtarget T210:=[[105.200094,123.174878,10.399975],[0.000000,0.000000,1.000000,0.000000],[0,0,-1,0],[9E+09,9E+09,9E+09,9E+09,9E+09,9E+09]];
    CONST robtarget T211:=[[105.200094,36.825129,10.399975],[0.000000,0.000000,1.000000,0.000000],[0,0,-1,0],[9E+09,9E+09,9E+09,9E+09,9E+09,9E+09]];
    CONST robtarget T212:=[[106.460098,37.589739,10.399975],[0.000000,0.000000,1.000000,0.000000],[0,0,-1,0],[9E+09,9E+09,9E+09,9E+09,9E+09,9E+09]];
    CONST robtarget T213:=[[106.460098,122.410268,10.399975],[0.000000,0.000000,1.000000,0.000000],[0,0,-1,0],[9E+09,9E+09,9E+09,9E+09,9E+09,9E+09]];
    CONST robtarget T214:=[[107.720103,121.607260,10.399975],[0.000000,0.000000,1.000000,0.000000],[0,0,-1,0],[9E+09,9E+09,9E+09,9E+09,9E+09,9E+09]];
    CONST robtarget T215:=[[107.720103,81.789524,10.399975],[0.000000,0.000000,1.000000,0.000000],[0,0,-1,0],[9E+09,9E+09,9E+09,9E+09,9E+09,9E+09]];
    CONST robtarget T216:=[[107.720103,78.210483,10.399975],[0.000000,0.000000,1.000000,0.000000],[0,0,-1,0],[9E+09,9E+09,9E+09,9E+09,9E+09,9E+09]];
    CONST robtarget T217:=[[107.720103,38.392748,10.399975],[0.000000,0.000000,1.000000,0.000000],[0,0,-1,0],[9E+09,9E+09,9E+09,9E+09,9E+09,9E+09]];
    CONST robtarget T218:=[[108.980107,39.265681,10.399975],[0.000000,0.000000,1.000000,0.000000],[0,0,-1,0],[9E+09,9E+09,9E+09,9E+09,9E+09,9E+09]];
    CONST robtarget T219:=[[108.980107,75.547902,10.399975],[0.000000,0.000000,1.000000,0.000000],[0,0,-1,0],[9E+09,9E+09,9E+09,9E+09,9E+09,9E+09]];
    CONST robtarget T220:=[[108.980107,84.452106,10.399975],[0.000000,0.000000,1.000000,0.000000],[0,0,-1,0],[9E+09,9E+09,9E+09,9E+09,9E+09,9E+09]];
    CONST robtarget T221:=[[108.980107,120.734326,10.399975],[0.000000,0.000000,1.000000,0.000000],[0,0,-1,0],[9E+09,9E+09,9E+09,9E+09,9E+09,9E+09]];
    CONST robtarget T222:=[[110.240112,119.803025,10.399975],[0.000000,0.000000,1.000000,0.000000],[0,0,-1,0],[9E+09,9E+09,9E+09,9E+09,9E+09,9E+09]];
    CONST robtarget T223:=[[110.240112,85.779969,10.399975],[0.000000,0.000000,1.000000,0.000000],[0,0,-1,0],[9E+09,9E+09,9E+09,9E+09,9E+09,9E+09]];
    CONST robtarget T224:=[[110.240112,74.220038,10.399975],[0.000000,0.000000,1.000000,0.000000],[0,0,-1,0],[9E+09,9E+09,9E+09,9E+09,9E+09,9E+09]];
    CONST robtarget T225:=[[110.240112,40.196983,10.399975],[0.000000,0.000000,1.000000,0.000000],[0,0,-1,0],[9E+09,9E+09,9E+09,9E+09,9E+09,9E+09]];
    CONST robtarget T226:=[[111.500116,41.180273,10.399975],[0.000000,0.000000,1.000000,0.000000],[0,0,-1,0],[9E+09,9E+09,9E+09,9E+09,9E+09,9E+09]];
    CONST robtarget T227:=[[111.500116,73.379202,10.399975],[0.000000,0.000000,1.000000,0.000000],[0,0,-1,0],[9E+09,9E+09,9E+09,9E+09,9E+09,9E+09]];
    CONST robtarget T228:=[[111.500116,86.620805,10.399975],[0.000000,0.000000,1.000000,0.000000],[0,0,-1,0],[9E+09,9E+09,9E+09,9E+09,9E+09,9E+09]];
    CONST robtarget T229:=[[111.500116,118.819735,10.399975],[0.000000,0.000000,1.000000,0.000000],[0,0,-1,0],[9E+09,9E+09,9E+09,9E+09,9E+09,9E+09]];
    CONST robtarget T230:=[[112.760121,117.767805,10.399975],[0.000000,0.000000,1.000000,0.000000],[0,0,-1,0],[9E+09,9E+09,9E+09,9E+09,9E+09,9E+09]];
    CONST robtarget T231:=[[112.760121,87.152583,10.399975],[0.000000,0.000000,1.000000,0.000000],[0,0,-1,0],[9E+09,9E+09,9E+09,9E+09,9E+09,9E+09]];
    CONST robtarget T232:=[[112.760121,72.847425,10.399975],[0.000000,0.000000,1.000000,0.000000],[0,0,-1,0],[9E+09,9E+09,9E+09,9E+09,9E+09,9E+09]];
    CONST robtarget T233:=[[112.760121,42.232203,10.399975],[0.000000,0.000000,1.000000,0.000000],[0,0,-1,0],[9E+09,9E+09,9E+09,9E+09,9E+09,9E+09]];
    CONST robtarget T234:=[[114.020125,43.373063,10.399975],[0.000000,0.000000,1.000000,0.000000],[0,0,-1,0],[9E+09,9E+09,9E+09,9E+09,9E+09,9E+09]];
    CONST robtarget T235:=[[114.020125,72.576253,10.399975],[0.000000,0.000000,1.000000,0.000000],[0,0,-1,0],[9E+09,9E+09,9E+09,9E+09,9E+09,9E+09]];
    CONST robtarget T236:=[[114.020125,87.423755,10.399975],[0.000000,0.000000,1.000000,0.000000],[0,0,-1,0],[9E+09,9E+09,9E+09,9E+09,9E+09,9E+09]];
    CONST robtarget T237:=[[114.020125,116.626944,10.399975],[0.000000,0.000000,1.000000,0.000000],[0,0,-1,0],[9E+09,9E+09,9E+09,9E+09,9E+09,9E+09]];
    CONST robtarget T238:=[[115.280130,115.412758,10.399975],[0.000000,0.000000,1.000000,0.000000],[0,0,-1,0],[9E+09,9E+09,9E+09,9E+09,9E+09,9E+09]];
    CONST robtarget T239:=[[115.280130,87.487316,10.399975],[0.000000,0.000000,1.000000,0.000000],[0,0,-1,0],[9E+09,9E+09,9E+09,9E+09,9E+09,9E+09]];
    CONST robtarget T240:=[[115.280130,72.512692,10.399975],[0.000000,0.000000,1.000000,0.000000],[0,0,-1,0],[9E+09,9E+09,9E+09,9E+09,9E+09,9E+09]];
    CONST robtarget T241:=[[115.280130,44.587250,10.399975],[0.000000,0.000000,1.000000,0.000000],[0,0,-1,0],[9E+09,9E+09,9E+09,9E+09,9E+09,9E+09]];
    CONST robtarget T242:=[[116.540134,45.884908,10.399975],[0.000000,0.000000,1.000000,0.000000],[0,0,-1,0],[9E+09,9E+09,9E+09,9E+09,9E+09,9E+09]];
    CONST robtarget T243:=[[116.540134,72.670297,10.399975],[0.000000,0.000000,1.000000,0.000000],[0,0,-1,0],[9E+09,9E+09,9E+09,9E+09,9E+09,9E+09]];
    CONST robtarget T244:=[[116.540134,87.329711,10.399975],[0.000000,0.000000,1.000000,0.000000],[0,0,-1,0],[9E+09,9E+09,9E+09,9E+09,9E+09,9E+09]];
    CONST robtarget T245:=[[116.540134,114.115099,10.399975],[0.000000,0.000000,1.000000,0.000000],[0,0,-1,0],[9E+09,9E+09,9E+09,9E+09,9E+09,9E+09]];
    CONST robtarget T246:=[[117.800139,112.721391,10.399975],[0.000000,0.000000,1.000000,0.000000],[0,0,-1,0],[9E+09,9E+09,9E+09,9E+09,9E+09,9E+09]];
    CONST robtarget T247:=[[117.800139,86.948670,10.399975],[0.000000,0.000000,1.000000,0.000000],[0,0,-1,0],[9E+09,9E+09,9E+09,9E+09,9E+09,9E+09]];
    CONST robtarget T248:=[[117.800139,73.051337,10.399975],[0.000000,0.000000,1.000000,0.000000],[0,0,-1,0],[9E+09,9E+09,9E+09,9E+09,9E+09,9E+09]];
    CONST robtarget T249:=[[117.800139,47.278617,10.399975],[0.000000,0.000000,1.000000,0.000000],[0,0,-1,0],[9E+09,9E+09,9E+09,9E+09,9E+09,9E+09]];
    CONST robtarget T250:=[[119.060143,48.787854,10.399975],[0.000000,0.000000,1.000000,0.000000],[0,0,-1,0],[9E+09,9E+09,9E+09,9E+09,9E+09,9E+09]];
    CONST robtarget T251:=[[119.060143,73.708792,10.399975],[0.000000,0.000000,1.000000,0.000000],[0,0,-1,0],[9E+09,9E+09,9E+09,9E+09,9E+09,9E+09]];
    CONST robtarget T252:=[[119.060143,86.291215,10.399975],[0.000000,0.000000,1.000000,0.000000],[0,0,-1,0],[9E+09,9E+09,9E+09,9E+09,9E+09,9E+09]];
    CONST robtarget T253:=[[119.060143,111.212154,10.399975],[0.000000,0.000000,1.000000,0.000000],[0,0,-1,0],[9E+09,9E+09,9E+09,9E+09,9E+09,9E+09]];
    CONST robtarget T254:=[[120.320148,109.560940,10.399975],[0.000000,0.000000,1.000000,0.000000],[0,0,-1,0],[9E+09,9E+09,9E+09,9E+09,9E+09,9E+09]];
    CONST robtarget T255:=[[120.320148,85.271589,10.399975],[0.000000,0.000000,1.000000,0.000000],[0,0,-1,0],[9E+09,9E+09,9E+09,9E+09,9E+09,9E+09]];
    CONST robtarget T256:=[[120.320148,74.728418,10.399975],[0.000000,0.000000,1.000000,0.000000],[0,0,-1,0],[9E+09,9E+09,9E+09,9E+09,9E+09,9E+09]];
    CONST robtarget T257:=[[120.320148,50.439068,10.399975],[0.000000,0.000000,1.000000,0.000000],[0,0,-1,0],[9E+09,9E+09,9E+09,9E+09,9E+09,9E+09]];
    CONST robtarget T258:=[[121.580152,52.240778,10.399975],[0.000000,0.000000,1.000000,0.000000],[0,0,-1,0],[9E+09,9E+09,9E+09,9E+09,9E+09,9E+09]];
    CONST robtarget T259:=[[121.580152,76.422528,10.399975],[0.000000,0.000000,1.000000,0.000000],[0,0,-1,0],[9E+09,9E+09,9E+09,9E+09,9E+09,9E+09]];
    CONST robtarget T260:=[[121.580152,83.577479,10.399975],[0.000000,0.000000,1.000000,0.000000],[0,0,-1,0],[9E+09,9E+09,9E+09,9E+09,9E+09,9E+09]];
    CONST robtarget T261:=[[121.580152,107.759230,10.399975],[0.000000,0.000000,1.000000,0.000000],[0,0,-1,0],[9E+09,9E+09,9E+09,9E+09,9E+09,9E+09]];
    CONST robtarget T262:=[[122.840157,105.775934,10.399975],[0.000000,0.000000,1.000000,0.000000],[0,0,-1,0],[9E+09,9E+09,9E+09,9E+09,9E+09,9E+09]];
    CONST robtarget T263:=[[122.840157,54.224074,10.399975],[0.000000,0.000000,1.000000,0.000000],[0,0,-1,0],[9E+09,9E+09,9E+09,9E+09,9E+09,9E+09]];
    CONST robtarget T264:=[[124.100161,56.444690,10.399975],[0.000000,0.000000,1.000000,0.000000],[0,0,-1,0],[9E+09,9E+09,9E+09,9E+09,9E+09,9E+09]];
    CONST robtarget T265:=[[124.100161,103.555317,10.399975],[0.000000,0.000000,1.000000,0.000000],[0,0,-1,0],[9E+09,9E+09,9E+09,9E+09,9E+09,9E+09]];
    CONST robtarget T266:=[[125.360166,101.007928,10.399975],[0.000000,0.000000,1.000000,0.000000],[0,0,-1,0],[9E+09,9E+09,9E+09,9E+09,9E+09,9E+09]];
    CONST robtarget T267:=[[125.360166,58.992080,10.399975],[0.000000,0.000000,1.000000,0.000000],[0,0,-1,0],[9E+09,9E+09,9E+09,9E+09,9E+09,9E+09]];
    CONST robtarget T268:=[[126.620170,61.953657,10.399975],[0.000000,0.000000,1.000000,0.000000],[0,0,-1,0],[9E+09,9E+09,9E+09,9E+09,9E+09,9E+09]];
    CONST robtarget T269:=[[126.620170,98.046351,10.399975],[0.000000,0.000000,1.000000,0.000000],[0,0,-1,0],[9E+09,9E+09,9E+09,9E+09,9E+09,9E+09]];
    CONST robtarget T270:=[[127.880175,94.360756,10.399975],[0.000000,0.000000,1.000000,0.000000],[0,0,-1,0],[9E+09,9E+09,9E+09,9E+09,9E+09,9E+09]];
    CONST robtarget T271:=[[127.880175,65.639251,10.399975],[0.000000,0.000000,1.000000,0.000000],[0,0,-1,0],[9E+09,9E+09,9E+09,9E+09,9E+09,9E+09]];
    CONST robtarget T272:=[[129.140179,70.797151,10.399975],[0.000000,0.000000,1.000000,0.000000],[0,0,-1,0],[9E+09,9E+09,9E+09,9E+09,9E+09,9E+09]];
    CONST robtarget T273:=[[129.140179,89.202857,10.399975],[0.000000,0.000000,1.000000,0.000000],[0,0,-1,0],[9E+09,9E+09,9E+09,9E+09,9E+09,9E+09]];
    CONST robtarget T274:=[[129.140179,70.797151,11.099985],[0.000000,0.000000,1.000000,0.000000],[0,0,-1,0],[9E+09,9E+09,9E+09,9E+09,9E+09,9E+09]];
    CONST robtarget T275:=[[129.140179,89.202857,11.099985],[0.000000,0.000000,1.000000,0.000000],[0,0,-1,0],[9E+09,9E+09,9E+09,9E+09,9E+09,9E+09]];
    CONST robtarget T276:=[[129.140179,70.797151,11.099985],[0.000000,0.000000,1.000000,0.000000],[0,0,-1,0],[9E+09,9E+09,9E+09,9E+09,9E+09,9E+09]];
    CONST robtarget T277:=[[129.140179,89.202857,11.099985],[0.000000,0.000000,1.000000,0.000000],[0,0,-1,0],[9E+09,9E+09,9E+09,9E+09,9E+09,9E+09]];
    CONST robtarget T278:=[[127.880175,94.360756,11.099985],[0.000000,0.000000,1.000000,0.000000],[0,0,-1,0],[9E+09,9E+09,9E+09,9E+09,9E+09,9E+09]];
    CONST robtarget T279:=[[127.880175,65.639251,11.099985],[0.000000,0.000000,1.000000,0.000000],[0,0,-1,0],[9E+09,9E+09,9E+09,9E+09,9E+09,9E+09]];
    CONST robtarget T280:=[[126.620170,61.953657,11.099985],[0.000000,0.000000,1.000000,0.000000],[0,0,-1,0],[9E+09,9E+09,9E+09,9E+09,9E+09,9E+09]];
    CONST robtarget T281:=[[126.620170,98.046351,11.099985],[0.000000,0.000000,1.000000,0.000000],[0,0,-1,0],[9E+09,9E+09,9E+09,9E+09,9E+09,9E+09]];
    CONST robtarget T282:=[[125.360166,101.007928,11.099985],[0.000000,0.000000,1.000000,0.000000],[0,0,-1,0],[9E+09,9E+09,9E+09,9E+09,9E+09,9E+09]];
    CONST robtarget T283:=[[125.360166,58.992080,11.099985],[0.000000,0.000000,1.000000,0.000000],[0,0,-1,0],[9E+09,9E+09,9E+09,9E+09,9E+09,9E+09]];
    CONST robtarget T284:=[[124.100161,56.444690,11.099985],[0.000000,0.000000,1.000000,0.000000],[0,0,-1,0],[9E+09,9E+09,9E+09,9E+09,9E+09,9E+09]];
    CONST robtarget T285:=[[124.100161,103.555317,11.099985],[0.000000,0.000000,1.000000,0.000000],[0,0,-1,0],[9E+09,9E+09,9E+09,9E+09,9E+09,9E+09]];
    CONST robtarget T286:=[[122.840157,105.775934,11.099985],[0.000000,0.000000,1.000000,0.000000],[0,0,-1,0],[9E+09,9E+09,9E+09,9E+09,9E+09,9E+09]];
    CONST robtarget T287:=[[122.840157,54.224074,11.099985],[0.000000,0.000000,1.000000,0.000000],[0,0,-1,0],[9E+09,9E+09,9E+09,9E+09,9E+09,9E+09]];
    CONST robtarget T288:=[[121.580152,52.240778,11.099985],[0.000000,0.000000,1.000000,0.000000],[0,0,-1,0],[9E+09,9E+09,9E+09,9E+09,9E+09,9E+09]];
    CONST robtarget T289:=[[121.580152,76.422528,11.099985],[0.000000,0.000000,1.000000,0.000000],[0,0,-1,0],[9E+09,9E+09,9E+09,9E+09,9E+09,9E+09]];
    CONST robtarget T290:=[[121.580152,83.577479,11.099985],[0.000000,0.000000,1.000000,0.000000],[0,0,-1,0],[9E+09,9E+09,9E+09,9E+09,9E+09,9E+09]];
    CONST robtarget T291:=[[121.580152,107.759230,11.099985],[0.000000,0.000000,1.000000,0.000000],[0,0,-1,0],[9E+09,9E+09,9E+09,9E+09,9E+09,9E+09]];
    CONST robtarget T292:=[[120.320148,109.560940,11.099985],[0.000000,0.000000,1.000000,0.000000],[0,0,-1,0],[9E+09,9E+09,9E+09,9E+09,9E+09,9E+09]];
    CONST robtarget T293:=[[120.320148,85.271589,11.099985],[0.000000,0.000000,1.000000,0.000000],[0,0,-1,0],[9E+09,9E+09,9E+09,9E+09,9E+09,9E+09]];
    CONST robtarget T294:=[[120.320148,74.728418,11.099985],[0.000000,0.000000,1.000000,0.000000],[0,0,-1,0],[9E+09,9E+09,9E+09,9E+09,9E+09,9E+09]];
    CONST robtarget T295:=[[120.320148,50.439068,11.099985],[0.000000,0.000000,1.000000,0.000000],[0,0,-1,0],[9E+09,9E+09,9E+09,9E+09,9E+09,9E+09]];
    CONST robtarget T296:=[[119.060143,48.787854,11.099985],[0.000000,0.000000,1.000000,0.000000],[0,0,-1,0],[9E+09,9E+09,9E+09,9E+09,9E+09,9E+09]];
    CONST robtarget T297:=[[119.060143,73.708792,11.099985],[0.000000,0.000000,1.000000,0.000000],[0,0,-1,0],[9E+09,9E+09,9E+09,9E+09,9E+09,9E+09]];
    CONST robtarget T298:=[[119.060143,86.291215,11.099985],[0.000000,0.000000,1.000000,0.000000],[0,0,-1,0],[9E+09,9E+09,9E+09,9E+09,9E+09,9E+09]];
    CONST robtarget T299:=[[119.060143,111.212154,11.099985],[0.000000,0.000000,1.000000,0.000000],[0,0,-1,0],[9E+09,9E+09,9E+09,9E+09,9E+09,9E+09]];
    CONST robtarget T300:=[[117.800139,112.721391,11.099985],[0.000000,0.000000,1.000000,0.000000],[0,0,-1,0],[9E+09,9E+09,9E+09,9E+09,9E+09,9E+09]];
    CONST robtarget T301:=[[117.800139,86.948670,11.099985],[0.000000,0.000000,1.000000,0.000000],[0,0,-1,0],[9E+09,9E+09,9E+09,9E+09,9E+09,9E+09]];
    CONST robtarget T302:=[[117.800139,73.051337,11.099985],[0.000000,0.000000,1.000000,0.000000],[0,0,-1,0],[9E+09,9E+09,9E+09,9E+09,9E+09,9E+09]];
    CONST robtarget T303:=[[117.800139,47.278617,11.099985],[0.000000,0.000000,1.000000,0.000000],[0,0,-1,0],[9E+09,9E+09,9E+09,9E+09,9E+09,9E+09]];
    CONST robtarget T304:=[[116.540134,45.884908,11.099985],[0.000000,0.000000,1.000000,0.000000],[0,0,-1,0],[9E+09,9E+09,9E+09,9E+09,9E+09,9E+09]];
    CONST robtarget T305:=[[116.540134,72.670297,11.099985],[0.000000,0.000000,1.000000,0.000000],[0,0,-1,0],[9E+09,9E+09,9E+09,9E+09,9E+09,9E+09]];
    CONST robtarget T306:=[[116.540134,87.329711,11.099985],[0.000000,0.000000,1.000000,0.000000],[0,0,-1,0],[9E+09,9E+09,9E+09,9E+09,9E+09,9E+09]];
    CONST robtarget T307:=[[116.540134,114.115099,11.099985],[0.000000,0.000000,1.000000,0.000000],[0,0,-1,0],[9E+09,9E+09,9E+09,9E+09,9E+09,9E+09]];
    CONST robtarget T308:=[[115.280130,115.412758,11.099985],[0.000000,0.000000,1.000000,0.000000],[0,0,-1,0],[9E+09,9E+09,9E+09,9E+09,9E+09,9E+09]];
    CONST robtarget T309:=[[115.280130,87.487316,11.099985],[0.000000,0.000000,1.000000,0.000000],[0,0,-1,0],[9E+09,9E+09,9E+09,9E+09,9E+09,9E+09]];
    CONST robtarget T310:=[[115.280130,72.512692,11.099985],[0.000000,0.000000,1.000000,0.000000],[0,0,-1,0],[9E+09,9E+09,9E+09,9E+09,9E+09,9E+09]];
    CONST robtarget T311:=[[115.280130,44.587250,11.099985],[0.000000,0.000000,1.000000,0.000000],[0,0,-1,0],[9E+09,9E+09,9E+09,9E+09,9E+09,9E+09]];
    CONST robtarget T312:=[[114.020125,43.373063,11.099985],[0.000000,0.000000,1.000000,0.000000],[0,0,-1,0],[9E+09,9E+09,9E+09,9E+09,9E+09,9E+09]];
    CONST robtarget T313:=[[114.020125,72.576253,11.099985],[0.000000,0.000000,1.000000,0.000000],[0,0,-1,0],[9E+09,9E+09,9E+09,9E+09,9E+09,9E+09]];
    CONST robtarget T314:=[[114.020125,87.423755,11.099985],[0.000000,0.000000,1.000000,0.000000],[0,0,-1,0],[9E+09,9E+09,9E+09,9E+09,9E+09,9E+09]];
    CONST robtarget T315:=[[114.020125,116.626944,11.099985],[0.000000,0.000000,1.000000,0.000000],[0,0,-1,0],[9E+09,9E+09,9E+09,9E+09,9E+09,9E+09]];
    CONST robtarget T316:=[[112.760121,117.767805,11.099985],[0.000000,0.000000,1.000000,0.000000],[0,0,-1,0],[9E+09,9E+09,9E+09,9E+09,9E+09,9E+09]];
    CONST robtarget T317:=[[112.760121,87.152583,11.099985],[0.000000,0.000000,1.000000,0.000000],[0,0,-1,0],[9E+09,9E+09,9E+09,9E+09,9E+09,9E+09]];
    CONST robtarget T318:=[[112.760121,72.847425,11.099985],[0.000000,0.000000,1.000000,0.000000],[0,0,-1,0],[9E+09,9E+09,9E+09,9E+09,9E+09,9E+09]];
    CONST robtarget T319:=[[112.760121,42.232203,11.099985],[0.000000,0.000000,1.000000,0.000000],[0,0,-1,0],[9E+09,9E+09,9E+09,9E+09,9E+09,9E+09]];
    CONST robtarget T320:=[[111.500116,41.180273,11.099985],[0.000000,0.000000,1.000000,0.000000],[0,0,-1,0],[9E+09,9E+09,9E+09,9E+09,9E+09,9E+09]];
    CONST robtarget T321:=[[111.500116,73.379202,11.099985],[0.000000,0.000000,1.000000,0.000000],[0,0,-1,0],[9E+09,9E+09,9E+09,9E+09,9E+09,9E+09]];
    CONST robtarget T322:=[[111.500116,86.620805,11.099985],[0.000000,0.000000,1.000000,0.000000],[0,0,-1,0],[9E+09,9E+09,9E+09,9E+09,9E+09,9E+09]];
    CONST robtarget T323:=[[111.500116,118.819735,11.099985],[0.000000,0.000000,1.000000,0.000000],[0,0,-1,0],[9E+09,9E+09,9E+09,9E+09,9E+09,9E+09]];
    CONST robtarget T324:=[[110.240112,119.803025,11.099985],[0.000000,0.000000,1.000000,0.000000],[0,0,-1,0],[9E+09,9E+09,9E+09,9E+09,9E+09,9E+09]];
    CONST robtarget T325:=[[110.240112,85.779969,11.099985],[0.000000,0.000000,1.000000,0.000000],[0,0,-1,0],[9E+09,9E+09,9E+09,9E+09,9E+09,9E+09]];
    CONST robtarget T326:=[[110.240112,74.220038,11.099985],[0.000000,0.000000,1.000000,0.000000],[0,0,-1,0],[9E+09,9E+09,9E+09,9E+09,9E+09,9E+09]];
    CONST robtarget T327:=[[110.240112,40.196983,11.099985],[0.000000,0.000000,1.000000,0.000000],[0,0,-1,0],[9E+09,9E+09,9E+09,9E+09,9E+09,9E+09]];
    CONST robtarget T328:=[[108.980107,39.265681,11.099985],[0.000000,0.000000,1.000000,0.000000],[0,0,-1,0],[9E+09,9E+09,9E+09,9E+09,9E+09,9E+09]];
    CONST robtarget T329:=[[108.980107,75.547902,11.099985],[0.000000,0.000000,1.000000,0.000000],[0,0,-1,0],[9E+09,9E+09,9E+09,9E+09,9E+09,9E+09]];
    CONST robtarget T330:=[[108.980107,84.452106,11.099985],[0.000000,0.000000,1.000000,0.000000],[0,0,-1,0],[9E+09,9E+09,9E+09,9E+09,9E+09,9E+09]];
    CONST robtarget T331:=[[108.980107,120.734326,11.099985],[0.000000,0.000000,1.000000,0.000000],[0,0,-1,0],[9E+09,9E+09,9E+09,9E+09,9E+09,9E+09]];
    CONST robtarget T332:=[[107.720103,121.607260,11.099985],[0.000000,0.000000,1.000000,0.000000],[0,0,-1,0],[9E+09,9E+09,9E+09,9E+09,9E+09,9E+09]];
    CONST robtarget T333:=[[107.720103,81.789524,11.099985],[0.000000,0.000000,1.000000,0.000000],[0,0,-1,0],[9E+09,9E+09,9E+09,9E+09,9E+09,9E+09]];
    CONST robtarget T334:=[[107.720103,78.210483,11.099985],[0.000000,0.000000,1.000000,0.000000],[0,0,-1,0],[9E+09,9E+09,9E+09,9E+09,9E+09,9E+09]];
    CONST robtarget T335:=[[107.720103,38.392748,11.099985],[0.000000,0.000000,1.000000,0.000000],[0,0,-1,0],[9E+09,9E+09,9E+09,9E+09,9E+09,9E+09]];
    CONST robtarget T336:=[[106.460098,37.589739,11.099985],[0.000000,0.000000,1.000000,0.000000],[0,0,-1,0],[9E+09,9E+09,9E+09,9E+09,9E+09,9E+09]];
    CONST robtarget T337:=[[106.460098,122.410268,11.099985],[0.000000,0.000000,1.000000,0.000000],[0,0,-1,0],[9E+09,9E+09,9E+09,9E+09,9E+09,9E+09]];
    CONST robtarget T338:=[[105.200094,123.174878,11.099985],[0.000000,0.000000,1.000000,0.000000],[0,0,-1,0],[9E+09,9E+09,9E+09,9E+09,9E+09,9E+09]];
    CONST robtarget T339:=[[105.200094,36.825129,11.099985],[0.000000,0.000000,1.000000,0.000000],[0,0,-1,0],[9E+09,9E+09,9E+09,9E+09,9E+09,9E+09]];
    CONST robtarget T340:=[[103.940089,36.110177,11.099985],[0.000000,0.000000,1.000000,0.000000],[0,0,-1,0],[9E+09,9E+09,9E+09,9E+09,9E+09,9E+09]];
    CONST robtarget T341:=[[103.940089,123.889831,11.099985],[0.000000,0.000000,1.000000,0.000000],[0,0,-1,0],[9E+09,9E+09,9E+09,9E+09,9E+09,9E+09]];
    CONST robtarget T342:=[[102.680085,124.546114,11.099985],[0.000000,0.000000,1.000000,0.000000],[0,0,-1,0],[9E+09,9E+09,9E+09,9E+09,9E+09,9E+09]];
    CONST robtarget T343:=[[102.680085,35.453894,11.099985],[0.000000,0.000000,1.000000,0.000000],[0,0,-1,0],[9E+09,9E+09,9E+09,9E+09,9E+09,9E+09]];
    CONST robtarget T344:=[[101.420080,34.827050,11.099985],[0.000000,0.000000,1.000000,0.000000],[0,0,-1,0],[9E+09,9E+09,9E+09,9E+09,9E+09,9E+09]];
    CONST robtarget T345:=[[101.420080,125.172958,11.099985],[0.000000,0.000000,1.000000,0.000000],[0,0,-1,0],[9E+09,9E+09,9E+09,9E+09,9E+09,9E+09]];
    CONST robtarget T346:=[[100.160076,125.745278,11.099985],[0.000000,0.000000,1.000000,0.000000],[0,0,-1,0],[9E+09,9E+09,9E+09,9E+09,9E+09,9E+09]];
    CONST robtarget T347:=[[100.160076,34.254730,11.099985],[0.000000,0.000000,1.000000,0.000000],[0,0,-1,0],[9E+09,9E+09,9E+09,9E+09,9E+09,9E+09]];
    CONST robtarget T348:=[[98.900071,33.722290,11.099985],[0.000000,0.000000,1.000000,0.000000],[0,0,-1,0],[9E+09,9E+09,9E+09,9E+09,9E+09,9E+09]];
    CONST robtarget T349:=[[98.900071,126.277717,11.099985],[0.000000,0.000000,1.000000,0.000000],[0,0,-1,0],[9E+09,9E+09,9E+09,9E+09,9E+09,9E+09]];
    CONST robtarget T350:=[[97.640067,126.783143,11.099985],[0.000000,0.000000,1.000000,0.000000],[0,0,-1,0],[9E+09,9E+09,9E+09,9E+09,9E+09,9E+09]];
    CONST robtarget T351:=[[97.640067,33.216864,11.099985],[0.000000,0.000000,1.000000,0.000000],[0,0,-1,0],[9E+09,9E+09,9E+09,9E+09,9E+09,9E+09]];
    CONST robtarget T352:=[[96.380062,32.772318,11.099985],[0.000000,0.000000,1.000000,0.000000],[0,0,-1,0],[9E+09,9E+09,9E+09,9E+09,9E+09,9E+09]];
    CONST robtarget T353:=[[96.380062,127.227690,11.099985],[0.000000,0.000000,1.000000,0.000000],[0,0,-1,0],[9E+09,9E+09,9E+09,9E+09,9E+09,9E+09]];
    CONST robtarget T354:=[[95.120058,127.652167,11.099985],[0.000000,0.000000,1.000000,0.000000],[0,0,-1,0],[9E+09,9E+09,9E+09,9E+09,9E+09,9E+09]];
    CONST robtarget T355:=[[95.120058,32.347841,11.099985],[0.000000,0.000000,1.000000,0.000000],[0,0,-1,0],[9E+09,9E+09,9E+09,9E+09,9E+09,9E+09]];
    CONST robtarget T356:=[[93.860053,31.969479,11.099985],[0.000000,0.000000,1.000000,0.000000],[0,0,-1,0],[9E+09,9E+09,9E+09,9E+09,9E+09,9E+09]];
    CONST robtarget T357:=[[93.860053,128.030529,11.099985],[0.000000,0.000000,1.000000,0.000000],[0,0,-1,0],[9E+09,9E+09,9E+09,9E+09,9E+09,9E+09]];
    CONST robtarget T358:=[[92.600049,128.374988,11.099985],[0.000000,0.000000,1.000000,0.000000],[0,0,-1,0],[9E+09,9E+09,9E+09,9E+09,9E+09,9E+09]];
    CONST robtarget T359:=[[92.600049,31.625019,11.099985],[0.000000,0.000000,1.000000,0.000000],[0,0,-1,0],[9E+09,9E+09,9E+09,9E+09,9E+09,9E+09]];
    CONST robtarget T360:=[[91.340044,31.307526,11.099985],[0.000000,0.000000,1.000000,0.000000],[0,0,-1,0],[9E+09,9E+09,9E+09,9E+09,9E+09,9E+09]];
    CONST robtarget T361:=[[91.340044,128.692481,11.099985],[0.000000,0.000000,1.000000,0.000000],[0,0,-1,0],[9E+09,9E+09,9E+09,9E+09,9E+09,9E+09]];
    CONST robtarget T362:=[[90.080040,128.960575,11.099985],[0.000000,0.000000,1.000000,0.000000],[0,0,-1,0],[9E+09,9E+09,9E+09,9E+09,9E+09,9E+09]];
    CONST robtarget T363:=[[90.080040,31.039433,11.099985],[0.000000,0.000000,1.000000,0.000000],[0,0,-1,0],[9E+09,9E+09,9E+09,9E+09,9E+09,9E+09]];
    CONST robtarget T364:=[[88.820035,30.786444,11.099985],[0.000000,0.000000,1.000000,0.000000],[0,0,-1,0],[9E+09,9E+09,9E+09,9E+09,9E+09,9E+09]];
    CONST robtarget T365:=[[88.820035,129.213563,11.099985],[0.000000,0.000000,1.000000,0.000000],[0,0,-1,0],[9E+09,9E+09,9E+09,9E+09,9E+09,9E+09]];
    CONST robtarget T366:=[[87.560031,129.413129,11.099985],[0.000000,0.000000,1.000000,0.000000],[0,0,-1,0],[9E+09,9E+09,9E+09,9E+09,9E+09,9E+09]];
    CONST robtarget T367:=[[87.560031,30.586879,11.099985],[0.000000,0.000000,1.000000,0.000000],[0,0,-1,0],[9E+09,9E+09,9E+09,9E+09,9E+09,9E+09]];
    CONST robtarget T368:=[[86.300026,30.406130,11.099985],[0.000000,0.000000,1.000000,0.000000],[0,0,-1,0],[9E+09,9E+09,9E+09,9E+09,9E+09,9E+09]];
    CONST robtarget T369:=[[86.300026,40.937335,11.099985],[0.000000,0.000000,1.000000,0.000000],[0,0,-1,0],[9E+09,9E+09,9E+09,9E+09,9E+09,9E+09]];
    CONST robtarget T370:=[[86.300026,49.062665,11.099985],[0.000000,0.000000,1.000000,0.000000],[0,0,-1,0],[9E+09,9E+09,9E+09,9E+09,9E+09,9E+09]];
    CONST robtarget T371:=[[86.300026,75.937339,11.099985],[0.000000,0.000000,1.000000,0.000000],[0,0,-1,0],[9E+09,9E+09,9E+09,9E+09,9E+09,9E+09]];
    CONST robtarget T372:=[[86.300026,84.062668,11.099985],[0.000000,0.000000,1.000000,0.000000],[0,0,-1,0],[9E+09,9E+09,9E+09,9E+09,9E+09,9E+09]];
    CONST robtarget T373:=[[86.300026,110.937342,11.099985],[0.000000,0.000000,1.000000,0.000000],[0,0,-1,0],[9E+09,9E+09,9E+09,9E+09,9E+09,9E+09]];
    CONST robtarget T374:=[[86.300026,119.062672,11.099985],[0.000000,0.000000,1.000000,0.000000],[0,0,-1,0],[9E+09,9E+09,9E+09,9E+09,9E+09,9E+09]];
    CONST robtarget T375:=[[86.300026,129.593877,11.099985],[0.000000,0.000000,1.000000,0.000000],[0,0,-1,0],[9E+09,9E+09,9E+09,9E+09,9E+09,9E+09]];
    CONST robtarget T376:=[[85.040022,129.735844,11.099985],[0.000000,0.000000,1.000000,0.000000],[0,0,-1,0],[9E+09,9E+09,9E+09,9E+09,9E+09,9E+09]];
    CONST robtarget T377:=[[85.040022,120.544921,11.099985],[0.000000,0.000000,1.000000,0.000000],[0,0,-1,0],[9E+09,9E+09,9E+09,9E+09,9E+09,9E+09]];
    CONST robtarget T378:=[[85.040022,109.455091,11.099985],[0.000000,0.000000,1.000000,0.000000],[0,0,-1,0],[9E+09,9E+09,9E+09,9E+09,9E+09,9E+09]];
    CONST robtarget T379:=[[85.040022,85.544918,11.099985],[0.000000,0.000000,1.000000,0.000000],[0,0,-1,0],[9E+09,9E+09,9E+09,9E+09,9E+09,9E+09]];
    CONST robtarget T380:=[[85.040022,74.455090,11.099985],[0.000000,0.000000,1.000000,0.000000],[0,0,-1,0],[9E+09,9E+09,9E+09,9E+09,9E+09,9E+09]];
    CONST robtarget T381:=[[85.040022,50.544916,11.099985],[0.000000,0.000000,1.000000,0.000000],[0,0,-1,0],[9E+09,9E+09,9E+09,9E+09,9E+09,9E+09]];
    CONST robtarget T382:=[[85.040022,39.455086,11.099985],[0.000000,0.000000,1.000000,0.000000],[0,0,-1,0],[9E+09,9E+09,9E+09,9E+09,9E+09,9E+09]];
    CONST robtarget T383:=[[85.040022,30.264163,11.099985],[0.000000,0.000000,1.000000,0.000000],[0,0,-1,0],[9E+09,9E+09,9E+09,9E+09,9E+09,9E+09]];
    CONST robtarget T384:=[[83.780017,30.153959,11.099985],[0.000000,0.000000,1.000000,0.000000],[0,0,-1,0],[9E+09,9E+09,9E+09,9E+09,9E+09,9E+09]];
    CONST robtarget T385:=[[83.780017,38.524551,11.099985],[0.000000,0.000000,1.000000,0.000000],[0,0,-1,0],[9E+09,9E+09,9E+09,9E+09,9E+09,9E+09]];
    CONST robtarget T386:=[[83.780017,51.475451,11.099985],[0.000000,0.000000,1.000000,0.000000],[0,0,-1,0],[9E+09,9E+09,9E+09,9E+09,9E+09,9E+09]];
    CONST robtarget T387:=[[83.780017,73.524553,11.099985],[0.000000,0.000000,1.000000,0.000000],[0,0,-1,0],[9E+09,9E+09,9E+09,9E+09,9E+09,9E+09]];
    CONST robtarget T388:=[[83.780017,86.475455,11.099985],[0.000000,0.000000,1.000000,0.000000],[0,0,-1,0],[9E+09,9E+09,9E+09,9E+09,9E+09,9E+09]];
    CONST robtarget T389:=[[83.780017,108.524556,11.099985],[0.000000,0.000000,1.000000,0.000000],[0,0,-1,0],[9E+09,9E+09,9E+09,9E+09,9E+09,9E+09]];
    CONST robtarget T390:=[[83.780017,121.475457,11.099985],[0.000000,0.000000,1.000000,0.000000],[0,0,-1,0],[9E+09,9E+09,9E+09,9E+09,9E+09,9E+09]];
    CONST robtarget T391:=[[83.780017,129.846049,11.099985],[0.000000,0.000000,1.000000,0.000000],[0,0,-1,0],[9E+09,9E+09,9E+09,9E+09,9E+09,9E+09]];
    CONST robtarget T392:=[[82.520013,129.931001,11.099985],[0.000000,0.000000,1.000000,0.000000],[0,0,-1,0],[9E+09,9E+09,9E+09,9E+09,9E+09,9E+09]];
    CONST robtarget T393:=[[82.520013,122.050628,11.099985],[0.000000,0.000000,1.000000,0.000000],[0,0,-1,0],[9E+09,9E+09,9E+09,9E+09,9E+09,9E+09]];
    CONST robtarget T394:=[[82.520013,107.949384,11.099985],[0.000000,0.000000,1.000000,0.000000],[0,0,-1,0],[9E+09,9E+09,9E+09,9E+09,9E+09,9E+09]];
    CONST robtarget T395:=[[82.520013,87.050626,11.099985],[0.000000,0.000000,1.000000,0.000000],[0,0,-1,0],[9E+09,9E+09,9E+09,9E+09,9E+09,9E+09]];
    CONST robtarget T396:=[[82.520013,72.949381,11.099985],[0.000000,0.000000,1.000000,0.000000],[0,0,-1,0],[9E+09,9E+09,9E+09,9E+09,9E+09,9E+09]];
    CONST robtarget T397:=[[82.520013,52.050624,11.099985],[0.000000,0.000000,1.000000,0.000000],[0,0,-1,0],[9E+09,9E+09,9E+09,9E+09,9E+09,9E+09]];
    CONST robtarget T398:=[[82.520013,37.949379,11.099985],[0.000000,0.000000,1.000000,0.000000],[0,0,-1,0],[9E+09,9E+09,9E+09,9E+09,9E+09,9E+09]];
    CONST robtarget T399:=[[82.520013,30.069007,11.099985],[0.000000,0.000000,1.000000,0.000000],[0,0,-1,0],[9E+09,9E+09,9E+09,9E+09,9E+09,9E+09]];
    CONST robtarget T400:=[[81.260008,30.028279,11.099985],[0.000000,0.000000,1.000000,0.000000],[0,0,-1,0],[9E+09,9E+09,9E+09,9E+09,9E+09,9E+09]];
    CONST robtarget T401:=[[81.260008,37.608991,11.099985],[0.000000,0.000000,1.000000,0.000000],[0,0,-1,0],[9E+09,9E+09,9E+09,9E+09,9E+09,9E+09]];
    CONST robtarget T402:=[[81.260008,52.391011,11.099985],[0.000000,0.000000,1.000000,0.000000],[0,0,-1,0],[9E+09,9E+09,9E+09,9E+09,9E+09,9E+09]];
    CONST robtarget T403:=[[81.260008,72.608994,11.099985],[0.000000,0.000000,1.000000,0.000000],[0,0,-1,0],[9E+09,9E+09,9E+09,9E+09,9E+09,9E+09]];
    CONST robtarget T404:=[[81.260008,87.391014,11.099985],[0.000000,0.000000,1.000000,0.000000],[0,0,-1,0],[9E+09,9E+09,9E+09,9E+09,9E+09,9E+09]];
    CONST robtarget T405:=[[81.260008,107.608996,11.099985],[0.000000,0.000000,1.000000,0.000000],[0,0,-1,0],[9E+09,9E+09,9E+09,9E+09,9E+09,9E+09]];
    CONST robtarget T406:=[[81.260008,122.391017,11.099985],[0.000000,0.000000,1.000000,0.000000],[0,0,-1,0],[9E+09,9E+09,9E+09,9E+09,9E+09,9E+09]];
    CONST robtarget T407:=[[81.260008,129.971729,11.099985],[0.000000,0.000000,1.000000,0.000000],[0,0,-1,0],[9E+09,9E+09,9E+09,9E+09,9E+09,9E+09]];
    CONST robtarget T408:=[[80.000004,130.000008,11.099985],[0.000000,0.000000,1.000000,0.000000],[0,0,-1,0],[9E+09,9E+09,9E+09,9E+09,9E+09,9E+09]];
    CONST robtarget T409:=[[80.000004,122.487319,11.099985],[0.000000,0.000000,1.000000,0.000000],[0,0,-1,0],[9E+09,9E+09,9E+09,9E+09,9E+09,9E+09]];
    CONST robtarget T410:=[[80.000004,107.512696,11.099985],[0.000000,0.000000,1.000000,0.000000],[0,0,-1,0],[9E+09,9E+09,9E+09,9E+09,9E+09,9E+09]];
    CONST robtarget T411:=[[80.000004,87.487316,11.099985],[0.000000,0.000000,1.000000,0.000000],[0,0,-1,0],[9E+09,9E+09,9E+09,9E+09,9E+09,9E+09]];
    CONST robtarget T412:=[[80.000004,72.512692,11.099985],[0.000000,0.000000,1.000000,0.000000],[0,0,-1,0],[9E+09,9E+09,9E+09,9E+09,9E+09,9E+09]];
    CONST robtarget T413:=[[80.000004,52.487312,11.099985],[0.000000,0.000000,1.000000,0.000000],[0,0,-1,0],[9E+09,9E+09,9E+09,9E+09,9E+09,9E+09]];
    CONST robtarget T414:=[[80.000004,37.512688,11.099985],[0.000000,0.000000,1.000000,0.000000],[0,0,-1,0],[9E+09,9E+09,9E+09,9E+09,9E+09,9E+09]];
    CONST robtarget T415:=[[80.000004,30.000000,11.099985],[0.000000,0.000000,1.000000,0.000000],[0,0,-1,0],[9E+09,9E+09,9E+09,9E+09,9E+09,9E+09]];
    CONST robtarget T416:=[[78.739999,30.028279,11.099985],[0.000000,0.000000,1.000000,0.000000],[0,0,-1,0],[9E+09,9E+09,9E+09,9E+09,9E+09,9E+09]];
    CONST robtarget T417:=[[78.739999,37.608991,11.099985],[0.000000,0.000000,1.000000,0.000000],[0,0,-1,0],[9E+09,9E+09,9E+09,9E+09,9E+09,9E+09]];
    CONST robtarget T418:=[[78.739999,52.391011,11.099985],[0.000000,0.000000,1.000000,0.000000],[0,0,-1,0],[9E+09,9E+09,9E+09,9E+09,9E+09,9E+09]];
    CONST robtarget T419:=[[78.739999,72.608994,11.099985],[0.000000,0.000000,1.000000,0.000000],[0,0,-1,0],[9E+09,9E+09,9E+09,9E+09,9E+09,9E+09]];
    CONST robtarget T420:=[[78.739999,87.391014,11.099985],[0.000000,0.000000,1.000000,0.000000],[0,0,-1,0],[9E+09,9E+09,9E+09,9E+09,9E+09,9E+09]];
    CONST robtarget T421:=[[78.739999,107.608996,11.099985],[0.000000,0.000000,1.000000,0.000000],[0,0,-1,0],[9E+09,9E+09,9E+09,9E+09,9E+09,9E+09]];
    CONST robtarget T422:=[[78.739999,122.391017,11.099985],[0.000000,0.000000,1.000000,0.000000],[0,0,-1,0],[9E+09,9E+09,9E+09,9E+09,9E+09,9E+09]];
    CONST robtarget T423:=[[78.739999,129.971729,11.099985],[0.000000,0.000000,1.000000,0.000000],[0,0,-1,0],[9E+09,9E+09,9E+09,9E+09,9E+09,9E+09]];
    CONST robtarget T424:=[[77.479995,129.931001,11.099985],[0.000000,0.000000,1.000000,0.000000],[0,0,-1,0],[9E+09,9E+09,9E+09,9E+09,9E+09,9E+09]];
    CONST robtarget T425:=[[77.479995,122.050628,11.099985],[0.000000,0.000000,1.000000,0.000000],[0,0,-1,0],[9E+09,9E+09,9E+09,9E+09,9E+09,9E+09]];
    CONST robtarget T426:=[[77.479995,107.949384,11.099985],[0.000000,0.000000,1.000000,0.000000],[0,0,-1,0],[9E+09,9E+09,9E+09,9E+09,9E+09,9E+09]];
    CONST robtarget T427:=[[77.479995,87.050626,11.099985],[0.000000,0.000000,1.000000,0.000000],[0,0,-1,0],[9E+09,9E+09,9E+09,9E+09,9E+09,9E+09]];
    CONST robtarget T428:=[[77.479995,72.949381,11.099985],[0.000000,0.000000,1.000000,0.000000],[0,0,-1,0],[9E+09,9E+09,9E+09,9E+09,9E+09,9E+09]];
    CONST robtarget T429:=[[77.479995,52.050624,11.099985],[0.000000,0.000000,1.000000,0.000000],[0,0,-1,0],[9E+09,9E+09,9E+09,9E+09,9E+09,9E+09]];
    CONST robtarget T430:=[[77.479995,37.949379,11.099985],[0.000000,0.000000,1.000000,0.000000],[0,0,-1,0],[9E+09,9E+09,9E+09,9E+09,9E+09,9E+09]];
    CONST robtarget T431:=[[77.479995,30.069007,11.099985],[0.000000,0.000000,1.000000,0.000000],[0,0,-1,0],[9E+09,9E+09,9E+09,9E+09,9E+09,9E+09]];
    CONST robtarget T432:=[[76.219990,30.153959,11.099985],[0.000000,0.000000,1.000000,0.000000],[0,0,-1,0],[9E+09,9E+09,9E+09,9E+09,9E+09,9E+09]];
    CONST robtarget T433:=[[76.219990,38.524551,11.099985],[0.000000,0.000000,1.000000,0.000000],[0,0,-1,0],[9E+09,9E+09,9E+09,9E+09,9E+09,9E+09]];
    CONST robtarget T434:=[[76.219990,51.475451,11.099985],[0.000000,0.000000,1.000000,0.000000],[0,0,-1,0],[9E+09,9E+09,9E+09,9E+09,9E+09,9E+09]];
    CONST robtarget T435:=[[76.219990,73.524553,11.099985],[0.000000,0.000000,1.000000,0.000000],[0,0,-1,0],[9E+09,9E+09,9E+09,9E+09,9E+09,9E+09]];
    CONST robtarget T436:=[[76.219990,86.475455,11.099985],[0.000000,0.000000,1.000000,0.000000],[0,0,-1,0],[9E+09,9E+09,9E+09,9E+09,9E+09,9E+09]];
    CONST robtarget T437:=[[76.219990,108.524556,11.099985],[0.000000,0.000000,1.000000,0.000000],[0,0,-1,0],[9E+09,9E+09,9E+09,9E+09,9E+09,9E+09]];
    CONST robtarget T438:=[[76.219990,121.475457,11.099985],[0.000000,0.000000,1.000000,0.000000],[0,0,-1,0],[9E+09,9E+09,9E+09,9E+09,9E+09,9E+09]];
    CONST robtarget T439:=[[76.219990,129.846049,11.099985],[0.000000,0.000000,1.000000,0.000000],[0,0,-1,0],[9E+09,9E+09,9E+09,9E+09,9E+09,9E+09]];
    CONST robtarget T440:=[[74.959986,129.735844,11.099985],[0.000000,0.000000,1.000000,0.000000],[0,0,-1,0],[9E+09,9E+09,9E+09,9E+09,9E+09,9E+09]];
    CONST robtarget T441:=[[74.959986,120.544921,11.099985],[0.000000,0.000000,1.000000,0.000000],[0,0,-1,0],[9E+09,9E+09,9E+09,9E+09,9E+09,9E+09]];
    CONST robtarget T442:=[[74.959986,109.455091,11.099985],[0.000000,0.000000,1.000000,0.000000],[0,0,-1,0],[9E+09,9E+09,9E+09,9E+09,9E+09,9E+09]];
    CONST robtarget T443:=[[74.959986,85.544918,11.099985],[0.000000,0.000000,1.000000,0.000000],[0,0,-1,0],[9E+09,9E+09,9E+09,9E+09,9E+09,9E+09]];
    CONST robtarget T444:=[[74.959986,74.455090,11.099985],[0.000000,0.000000,1.000000,0.000000],[0,0,-1,0],[9E+09,9E+09,9E+09,9E+09,9E+09,9E+09]];
    CONST robtarget T445:=[[74.959986,50.544916,11.099985],[0.000000,0.000000,1.000000,0.000000],[0,0,-1,0],[9E+09,9E+09,9E+09,9E+09,9E+09,9E+09]];
    CONST robtarget T446:=[[74.959986,39.455086,11.099985],[0.000000,0.000000,1.000000,0.000000],[0,0,-1,0],[9E+09,9E+09,9E+09,9E+09,9E+09,9E+09]];
    CONST robtarget T447:=[[74.959986,30.264163,11.099985],[0.000000,0.000000,1.000000,0.000000],[0,0,-1,0],[9E+09,9E+09,9E+09,9E+09,9E+09,9E+09]];
    CONST robtarget T448:=[[73.699981,30.406130,11.099985],[0.000000,0.000000,1.000000,0.000000],[0,0,-1,0],[9E+09,9E+09,9E+09,9E+09,9E+09,9E+09]];
    CONST robtarget T449:=[[73.699981,40.937335,11.099985],[0.000000,0.000000,1.000000,0.000000],[0,0,-1,0],[9E+09,9E+09,9E+09,9E+09,9E+09,9E+09]];
    CONST robtarget T450:=[[73.699981,49.062665,11.099985],[0.000000,0.000000,1.000000,0.000000],[0,0,-1,0],[9E+09,9E+09,9E+09,9E+09,9E+09,9E+09]];
    CONST robtarget T451:=[[73.699981,75.937339,11.099985],[0.000000,0.000000,1.000000,0.000000],[0,0,-1,0],[9E+09,9E+09,9E+09,9E+09,9E+09,9E+09]];
    CONST robtarget T452:=[[73.699981,84.062668,11.099985],[0.000000,0.000000,1.000000,0.000000],[0,0,-1,0],[9E+09,9E+09,9E+09,9E+09,9E+09,9E+09]];
    CONST robtarget T453:=[[73.699981,110.937342,11.099985],[0.000000,0.000000,1.000000,0.000000],[0,0,-1,0],[9E+09,9E+09,9E+09,9E+09,9E+09,9E+09]];
    CONST robtarget T454:=[[73.699981,119.062672,11.099985],[0.000000,0.000000,1.000000,0.000000],[0,0,-1,0],[9E+09,9E+09,9E+09,9E+09,9E+09,9E+09]];
    CONST robtarget T455:=[[73.699981,129.593877,11.099985],[0.000000,0.000000,1.000000,0.000000],[0,0,-1,0],[9E+09,9E+09,9E+09,9E+09,9E+09,9E+09]];
    CONST robtarget T456:=[[72.439977,129.413129,11.099985],[0.000000,0.000000,1.000000,0.000000],[0,0,-1,0],[9E+09,9E+09,9E+09,9E+09,9E+09,9E+09]];
    CONST robtarget T457:=[[72.439977,30.586879,11.099985],[0.000000,0.000000,1.000000,0.000000],[0,0,-1,0],[9E+09,9E+09,9E+09,9E+09,9E+09,9E+09]];
    CONST robtarget T458:=[[71.179972,30.786444,11.099985],[0.000000,0.000000,1.000000,0.000000],[0,0,-1,0],[9E+09,9E+09,9E+09,9E+09,9E+09,9E+09]];
    CONST robtarget T459:=[[71.179972,129.213563,11.099985],[0.000000,0.000000,1.000000,0.000000],[0,0,-1,0],[9E+09,9E+09,9E+09,9E+09,9E+09,9E+09]];
    CONST robtarget T460:=[[69.919968,128.960575,11.099985],[0.000000,0.000000,1.000000,0.000000],[0,0,-1,0],[9E+09,9E+09,9E+09,9E+09,9E+09,9E+09]];
    CONST robtarget T461:=[[69.919968,31.039433,11.099985],[0.000000,0.000000,1.000000,0.000000],[0,0,-1,0],[9E+09,9E+09,9E+09,9E+09,9E+09,9E+09]];
    CONST robtarget T462:=[[68.659963,31.307526,11.099985],[0.000000,0.000000,1.000000,0.000000],[0,0,-1,0],[9E+09,9E+09,9E+09,9E+09,9E+09,9E+09]];
    CONST robtarget T463:=[[68.659963,128.692481,11.099985],[0.000000,0.000000,1.000000,0.000000],[0,0,-1,0],[9E+09,9E+09,9E+09,9E+09,9E+09,9E+09]];
    CONST robtarget T464:=[[67.399959,128.374988,11.099985],[0.000000,0.000000,1.000000,0.000000],[0,0,-1,0],[9E+09,9E+09,9E+09,9E+09,9E+09,9E+09]];
    CONST robtarget T465:=[[67.399959,31.625019,11.099985],[0.000000,0.000000,1.000000,0.000000],[0,0,-1,0],[9E+09,9E+09,9E+09,9E+09,9E+09,9E+09]];
    CONST robtarget T466:=[[66.139954,31.969479,11.099985],[0.000000,0.000000,1.000000,0.000000],[0,0,-1,0],[9E+09,9E+09,9E+09,9E+09,9E+09,9E+09]];
    CONST robtarget T467:=[[66.139954,128.030529,11.099985],[0.000000,0.000000,1.000000,0.000000],[0,0,-1,0],[9E+09,9E+09,9E+09,9E+09,9E+09,9E+09]];
    CONST robtarget T468:=[[64.879950,127.652167,11.099985],[0.000000,0.000000,1.000000,0.000000],[0,0,-1,0],[9E+09,9E+09,9E+09,9E+09,9E+09,9E+09]];
    CONST robtarget T469:=[[64.879950,32.347841,11.099985],[0.000000,0.000000,1.000000,0.000000],[0,0,-1,0],[9E+09,9E+09,9E+09,9E+09,9E+09,9E+09]];
    CONST robtarget T470:=[[63.619945,32.772318,11.099985],[0.000000,0.000000,1.000000,0.000000],[0,0,-1,0],[9E+09,9E+09,9E+09,9E+09,9E+09,9E+09]];
    CONST robtarget T471:=[[63.619945,127.227690,11.099985],[0.000000,0.000000,1.000000,0.000000],[0,0,-1,0],[9E+09,9E+09,9E+09,9E+09,9E+09,9E+09]];
    CONST robtarget T472:=[[62.359941,126.783143,11.099985],[0.000000,0.000000,1.000000,0.000000],[0,0,-1,0],[9E+09,9E+09,9E+09,9E+09,9E+09,9E+09]];
    CONST robtarget T473:=[[62.359941,33.216864,11.099985],[0.000000,0.000000,1.000000,0.000000],[0,0,-1,0],[9E+09,9E+09,9E+09,9E+09,9E+09,9E+09]];
    CONST robtarget T474:=[[61.099936,33.722290,11.099985],[0.000000,0.000000,1.000000,0.000000],[0,0,-1,0],[9E+09,9E+09,9E+09,9E+09,9E+09,9E+09]];
    CONST robtarget T475:=[[61.099936,126.277717,11.099985],[0.000000,0.000000,1.000000,0.000000],[0,0,-1,0],[9E+09,9E+09,9E+09,9E+09,9E+09,9E+09]];
    CONST robtarget T476:=[[59.839932,125.745278,11.099985],[0.000000,0.000000,1.000000,0.000000],[0,0,-1,0],[9E+09,9E+09,9E+09,9E+09,9E+09,9E+09]];
    CONST robtarget T477:=[[59.839932,34.254730,11.099985],[0.000000,0.000000,1.000000,0.000000],[0,0,-1,0],[9E+09,9E+09,9E+09,9E+09,9E+09,9E+09]];
    CONST robtarget T478:=[[58.579927,34.827050,11.099985],[0.000000,0.000000,1.000000,0.000000],[0,0,-1,0],[9E+09,9E+09,9E+09,9E+09,9E+09,9E+09]];
    CONST robtarget T479:=[[58.579927,125.172958,11.099985],[0.000000,0.000000,1.000000,0.000000],[0,0,-1,0],[9E+09,9E+09,9E+09,9E+09,9E+09,9E+09]];
    CONST robtarget T480:=[[57.319923,124.546114,11.099985],[0.000000,0.000000,1.000000,0.000000],[0,0,-1,0],[9E+09,9E+09,9E+09,9E+09,9E+09,9E+09]];
    CONST robtarget T481:=[[57.319923,35.453894,11.099985],[0.000000,0.000000,1.000000,0.000000],[0,0,-1,0],[9E+09,9E+09,9E+09,9E+09,9E+09,9E+09]];
    CONST robtarget T482:=[[56.059918,36.110177,11.099985],[0.000000,0.000000,1.000000,0.000000],[0,0,-1,0],[9E+09,9E+09,9E+09,9E+09,9E+09,9E+09]];
    CONST robtarget T483:=[[56.059918,123.889831,11.099985],[0.000000,0.000000,1.000000,0.000000],[0,0,-1,0],[9E+09,9E+09,9E+09,9E+09,9E+09,9E+09]];
    CONST robtarget T484:=[[54.799914,123.174878,11.099985],[0.000000,0.000000,1.000000,0.000000],[0,0,-1,0],[9E+09,9E+09,9E+09,9E+09,9E+09,9E+09]];
    CONST robtarget T485:=[[54.799914,36.825129,11.099985],[0.000000,0.000000,1.000000,0.000000],[0,0,-1,0],[9E+09,9E+09,9E+09,9E+09,9E+09,9E+09]];
    CONST robtarget T486:=[[53.539909,37.589739,11.099985],[0.000000,0.000000,1.000000,0.000000],[0,0,-1,0],[9E+09,9E+09,9E+09,9E+09,9E+09,9E+09]];
    CONST robtarget T487:=[[53.539909,122.410268,11.099985],[0.000000,0.000000,1.000000,0.000000],[0,0,-1,0],[9E+09,9E+09,9E+09,9E+09,9E+09,9E+09]];
    CONST robtarget T488:=[[52.279905,121.607260,11.099985],[0.000000,0.000000,1.000000,0.000000],[0,0,-1,0],[9E+09,9E+09,9E+09,9E+09,9E+09,9E+09]];
    CONST robtarget T489:=[[52.279905,81.789524,11.099985],[0.000000,0.000000,1.000000,0.000000],[0,0,-1,0],[9E+09,9E+09,9E+09,9E+09,9E+09,9E+09]];
    CONST robtarget T490:=[[52.279905,78.210483,11.099985],[0.000000,0.000000,1.000000,0.000000],[0,0,-1,0],[9E+09,9E+09,9E+09,9E+09,9E+09,9E+09]];
    CONST robtarget T491:=[[52.279905,38.392748,11.099985],[0.000000,0.000000,1.000000,0.000000],[0,0,-1,0],[9E+09,9E+09,9E+09,9E+09,9E+09,9E+09]];
    CONST robtarget T492:=[[51.019900,39.265681,11.099985],[0.000000,0.000000,1.000000,0.000000],[0,0,-1,0],[9E+09,9E+09,9E+09,9E+09,9E+09,9E+09]];
    CONST robtarget T493:=[[51.019900,75.547902,11.099985],[0.000000,0.000000,1.000000,0.000000],[0,0,-1,0],[9E+09,9E+09,9E+09,9E+09,9E+09,9E+09]];
    CONST robtarget T494:=[[51.019900,84.452106,11.099985],[0.000000,0.000000,1.000000,0.000000],[0,0,-1,0],[9E+09,9E+09,9E+09,9E+09,9E+09,9E+09]];
    CONST robtarget T495:=[[51.019900,120.734326,11.099985],[0.000000,0.000000,1.000000,0.000000],[0,0,-1,0],[9E+09,9E+09,9E+09,9E+09,9E+09,9E+09]];
    CONST robtarget T496:=[[49.759896,119.803025,11.099985],[0.000000,0.000000,1.000000,0.000000],[0,0,-1,0],[9E+09,9E+09,9E+09,9E+09,9E+09,9E+09]];
    CONST robtarget T497:=[[49.759896,85.779969,11.099985],[0.000000,0.000000,1.000000,0.000000],[0,0,-1,0],[9E+09,9E+09,9E+09,9E+09,9E+09,9E+09]];
    CONST robtarget T498:=[[49.759896,74.220038,11.099985],[0.000000,0.000000,1.000000,0.000000],[0,0,-1,0],[9E+09,9E+09,9E+09,9E+09,9E+09,9E+09]];
    CONST robtarget T499:=[[49.759896,40.196983,11.099985],[0.000000,0.000000,1.000000,0.000000],[0,0,-1,0],[9E+09,9E+09,9E+09,9E+09,9E+09,9E+09]];
    CONST robtarget T500:=[[48.499891,41.180273,11.099985],[0.000000,0.000000,1.000000,0.000000],[0,0,-1,0],[9E+09,9E+09,9E+09,9E+09,9E+09,9E+09]];
    CONST robtarget T501:=[[48.499891,73.379202,11.099985],[0.000000,0.000000,1.000000,0.000000],[0,0,-1,0],[9E+09,9E+09,9E+09,9E+09,9E+09,9E+09]];
    CONST robtarget T502:=[[48.499891,86.620805,11.099985],[0.000000,0.000000,1.000000,0.000000],[0,0,-1,0],[9E+09,9E+09,9E+09,9E+09,9E+09,9E+09]];
    CONST robtarget T503:=[[48.499891,118.819735,11.099985],[0.000000,0.000000,1.000000,0.000000],[0,0,-1,0],[9E+09,9E+09,9E+09,9E+09,9E+09,9E+09]];
    CONST robtarget T504:=[[47.239887,117.767805,11.099985],[0.000000,0.000000,1.000000,0.000000],[0,0,-1,0],[9E+09,9E+09,9E+09,9E+09,9E+09,9E+09]];
    CONST robtarget T505:=[[47.239887,87.152583,11.099985],[0.000000,0.000000,1.000000,0.000000],[0,0,-1,0],[9E+09,9E+09,9E+09,9E+09,9E+09,9E+09]];
    CONST robtarget T506:=[[47.239887,72.847425,11.099985],[0.000000,0.000000,1.000000,0.000000],[0,0,-1,0],[9E+09,9E+09,9E+09,9E+09,9E+09,9E+09]];
    CONST robtarget T507:=[[47.239887,42.232203,11.099985],[0.000000,0.000000,1.000000,0.000000],[0,0,-1,0],[9E+09,9E+09,9E+09,9E+09,9E+09,9E+09]];
    CONST robtarget T508:=[[45.979882,43.373063,11.099985],[0.000000,0.000000,1.000000,0.000000],[0,0,-1,0],[9E+09,9E+09,9E+09,9E+09,9E+09,9E+09]];
    CONST robtarget T509:=[[45.979882,72.576253,11.099985],[0.000000,0.000000,1.000000,0.000000],[0,0,-1,0],[9E+09,9E+09,9E+09,9E+09,9E+09,9E+09]];
    CONST robtarget T510:=[[45.979882,87.423755,11.099985],[0.000000,0.000000,1.000000,0.000000],[0,0,-1,0],[9E+09,9E+09,9E+09,9E+09,9E+09,9E+09]];
    CONST robtarget T511:=[[45.979882,116.626944,11.099985],[0.000000,0.000000,1.000000,0.000000],[0,0,-1,0],[9E+09,9E+09,9E+09,9E+09,9E+09,9E+09]];
    CONST robtarget T512:=[[44.719878,115.412758,11.099985],[0.000000,0.000000,1.000000,0.000000],[0,0,-1,0],[9E+09,9E+09,9E+09,9E+09,9E+09,9E+09]];
    CONST robtarget T513:=[[44.719878,87.487316,11.099985],[0.000000,0.000000,1.000000,0.000000],[0,0,-1,0],[9E+09,9E+09,9E+09,9E+09,9E+09,9E+09]];
    CONST robtarget T514:=[[44.719878,72.512692,11.099985],[0.000000,0.000000,1.000000,0.000000],[0,0,-1,0],[9E+09,9E+09,9E+09,9E+09,9E+09,9E+09]];
    CONST robtarget T515:=[[44.719878,44.587250,11.099985],[0.000000,0.000000,1.000000,0.000000],[0,0,-1,0],[9E+09,9E+09,9E+09,9E+09,9E+09,9E+09]];
    CONST robtarget T516:=[[43.459873,45.884908,11.099985],[0.000000,0.000000,1.000000,0.000000],[0,0,-1,0],[9E+09,9E+09,9E+09,9E+09,9E+09,9E+09]];
    CONST robtarget T517:=[[43.459873,72.670297,11.099985],[0.000000,0.000000,1.000000,0.000000],[0,0,-1,0],[9E+09,9E+09,9E+09,9E+09,9E+09,9E+09]];
    CONST robtarget T518:=[[43.459873,87.329711,11.099985],[0.000000,0.000000,1.000000,0.000000],[0,0,-1,0],[9E+09,9E+09,9E+09,9E+09,9E+09,9E+09]];
    CONST robtarget T519:=[[43.459873,114.115099,11.099985],[0.000000,0.000000,1.000000,0.000000],[0,0,-1,0],[9E+09,9E+09,9E+09,9E+09,9E+09,9E+09]];
    CONST robtarget T520:=[[42.199869,112.721391,11.099985],[0.000000,0.000000,1.000000,0.000000],[0,0,-1,0],[9E+09,9E+09,9E+09,9E+09,9E+09,9E+09]];
    CONST robtarget T521:=[[42.199869,86.948670,11.099985],[0.000000,0.000000,1.000000,0.000000],[0,0,-1,0],[9E+09,9E+09,9E+09,9E+09,9E+09,9E+09]];
    CONST robtarget T522:=[[42.199869,73.051337,11.099985],[0.000000,0.000000,1.000000,0.000000],[0,0,-1,0],[9E+09,9E+09,9E+09,9E+09,9E+09,9E+09]];
    CONST robtarget T523:=[[42.199869,47.278617,11.099985],[0.000000,0.000000,1.000000,0.000000],[0,0,-1,0],[9E+09,9E+09,9E+09,9E+09,9E+09,9E+09]];
    CONST robtarget T524:=[[40.939864,48.787854,11.099985],[0.000000,0.000000,1.000000,0.000000],[0,0,-1,0],[9E+09,9E+09,9E+09,9E+09,9E+09,9E+09]];
    CONST robtarget T525:=[[40.939864,73.708792,11.099985],[0.000000,0.000000,1.000000,0.000000],[0,0,-1,0],[9E+09,9E+09,9E+09,9E+09,9E+09,9E+09]];
    CONST robtarget T526:=[[40.939864,86.291215,11.099985],[0.000000,0.000000,1.000000,0.000000],[0,0,-1,0],[9E+09,9E+09,9E+09,9E+09,9E+09,9E+09]];
    CONST robtarget T527:=[[40.939864,111.212154,11.099985],[0.000000,0.000000,1.000000,0.000000],[0,0,-1,0],[9E+09,9E+09,9E+09,9E+09,9E+09,9E+09]];
    CONST robtarget T528:=[[39.679860,109.560940,11.099985],[0.000000,0.000000,1.000000,0.000000],[0,0,-1,0],[9E+09,9E+09,9E+09,9E+09,9E+09,9E+09]];
    CONST robtarget T529:=[[39.679860,85.271589,11.099985],[0.000000,0.000000,1.000000,0.000000],[0,0,-1,0],[9E+09,9E+09,9E+09,9E+09,9E+09,9E+09]];
    CONST robtarget T530:=[[39.679860,74.728418,11.099985],[0.000000,0.000000,1.000000,0.000000],[0,0,-1,0],[9E+09,9E+09,9E+09,9E+09,9E+09,9E+09]];
    CONST robtarget T531:=[[39.679860,50.439068,11.099985],[0.000000,0.000000,1.000000,0.000000],[0,0,-1,0],[9E+09,9E+09,9E+09,9E+09,9E+09,9E+09]];
    CONST robtarget T532:=[[38.419855,52.240778,11.099985],[0.000000,0.000000,1.000000,0.000000],[0,0,-1,0],[9E+09,9E+09,9E+09,9E+09,9E+09,9E+09]];
    CONST robtarget T533:=[[38.419855,76.422528,11.099985],[0.000000,0.000000,1.000000,0.000000],[0,0,-1,0],[9E+09,9E+09,9E+09,9E+09,9E+09,9E+09]];
    CONST robtarget T534:=[[38.419855,83.577479,11.099985],[0.000000,0.000000,1.000000,0.000000],[0,0,-1,0],[9E+09,9E+09,9E+09,9E+09,9E+09,9E+09]];
    CONST robtarget T535:=[[38.419855,107.759230,11.099985],[0.000000,0.000000,1.000000,0.000000],[0,0,-1,0],[9E+09,9E+09,9E+09,9E+09,9E+09,9E+09]];
    CONST robtarget T536:=[[37.159851,105.775934,11.099985],[0.000000,0.000000,1.000000,0.000000],[0,0,-1,0],[9E+09,9E+09,9E+09,9E+09,9E+09,9E+09]];
    CONST robtarget T537:=[[37.159851,54.224074,11.099985],[0.000000,0.000000,1.000000,0.000000],[0,0,-1,0],[9E+09,9E+09,9E+09,9E+09,9E+09,9E+09]];
    CONST robtarget T538:=[[35.899846,56.444690,11.099985],[0.000000,0.000000,1.000000,0.000000],[0,0,-1,0],[9E+09,9E+09,9E+09,9E+09,9E+09,9E+09]];
    CONST robtarget T539:=[[35.899846,103.555317,11.099985],[0.000000,0.000000,1.000000,0.000000],[0,0,-1,0],[9E+09,9E+09,9E+09,9E+09,9E+09,9E+09]];
    CONST robtarget T540:=[[34.639842,101.007928,11.099985],[0.000000,0.000000,1.000000,0.000000],[0,0,-1,0],[9E+09,9E+09,9E+09,9E+09,9E+09,9E+09]];
    CONST robtarget T541:=[[34.639842,58.992080,11.099985],[0.000000,0.000000,1.000000,0.000000],[0,0,-1,0],[9E+09,9E+09,9E+09,9E+09,9E+09,9E+09]];
    CONST robtarget T542:=[[33.379837,61.953657,11.099985],[0.000000,0.000000,1.000000,0.000000],[0,0,-1,0],[9E+09,9E+09,9E+09,9E+09,9E+09,9E+09]];
    CONST robtarget T543:=[[33.379837,98.046351,11.099985],[0.000000,0.000000,1.000000,0.000000],[0,0,-1,0],[9E+09,9E+09,9E+09,9E+09,9E+09,9E+09]];
    CONST robtarget T544:=[[32.119833,94.360756,11.099985],[0.000000,0.000000,1.000000,0.000000],[0,0,-1,0],[9E+09,9E+09,9E+09,9E+09,9E+09,9E+09]];
    CONST robtarget T545:=[[32.119833,65.639251,11.099985],[0.000000,0.000000,1.000000,0.000000],[0,0,-1,0],[9E+09,9E+09,9E+09,9E+09,9E+09,9E+09]];
    CONST robtarget T546:=[[30.859828,70.797151,11.099985],[0.000000,0.000000,1.000000,0.000000],[0,0,-1,0],[9E+09,9E+09,9E+09,9E+09,9E+09,9E+09]];
    CONST robtarget T547:=[[30.859828,89.202857,11.099985],[0.000000,0.000000,1.000000,0.000000],[0,0,-1,0],[9E+09,9E+09,9E+09,9E+09,9E+09,9E+09]];
    CONST robtarget T548:=[[30.859828,70.797151,11.799995],[0.000000,0.000000,1.000000,0.000000],[0,0,-1,0],[9E+09,9E+09,9E+09,9E+09,9E+09,9E+09]];
    CONST robtarget T549:=[[30.859828,89.202857,11.799995],[0.000000,0.000000,1.000000,0.000000],[0,0,-1,0],[9E+09,9E+09,9E+09,9E+09,9E+09,9E+09]];
    CONST robtarget T550:=[[30.859828,70.797151,11.799995],[0.000000,0.000000,1.000000,0.000000],[0,0,-1,0],[9E+09,9E+09,9E+09,9E+09,9E+09,9E+09]];
    CONST robtarget T551:=[[30.859828,89.202857,11.799995],[0.000000,0.000000,1.000000,0.000000],[0,0,-1,0],[9E+09,9E+09,9E+09,9E+09,9E+09,9E+09]];
    CONST robtarget T552:=[[32.119833,94.360756,11.799995],[0.000000,0.000000,1.000000,0.000000],[0,0,-1,0],[9E+09,9E+09,9E+09,9E+09,9E+09,9E+09]];
    CONST robtarget T553:=[[32.119833,65.639251,11.799995],[0.000000,0.000000,1.000000,0.000000],[0,0,-1,0],[9E+09,9E+09,9E+09,9E+09,9E+09,9E+09]];
    CONST robtarget T554:=[[33.379837,61.953657,11.799995],[0.000000,0.000000,1.000000,0.000000],[0,0,-1,0],[9E+09,9E+09,9E+09,9E+09,9E+09,9E+09]];
    CONST robtarget T555:=[[33.379837,98.046351,11.799995],[0.000000,0.000000,1.000000,0.000000],[0,0,-1,0],[9E+09,9E+09,9E+09,9E+09,9E+09,9E+09]];
    CONST robtarget T556:=[[34.639842,101.007928,11.799995],[0.000000,0.000000,1.000000,0.000000],[0,0,-1,0],[9E+09,9E+09,9E+09,9E+09,9E+09,9E+09]];
    CONST robtarget T557:=[[34.639842,58.992080,11.799995],[0.000000,0.000000,1.000000,0.000000],[0,0,-1,0],[9E+09,9E+09,9E+09,9E+09,9E+09,9E+09]];
    CONST robtarget T558:=[[35.899846,56.444690,11.799995],[0.000000,0.000000,1.000000,0.000000],[0,0,-1,0],[9E+09,9E+09,9E+09,9E+09,9E+09,9E+09]];
    CONST robtarget T559:=[[35.899846,103.555317,11.799995],[0.000000,0.000000,1.000000,0.000000],[0,0,-1,0],[9E+09,9E+09,9E+09,9E+09,9E+09,9E+09]];
    CONST robtarget T560:=[[37.159851,105.775934,11.799995],[0.000000,0.000000,1.000000,0.000000],[0,0,-1,0],[9E+09,9E+09,9E+09,9E+09,9E+09,9E+09]];
    CONST robtarget T561:=[[37.159851,54.224074,11.799995],[0.000000,0.000000,1.000000,0.000000],[0,0,-1,0],[9E+09,9E+09,9E+09,9E+09,9E+09,9E+09]];
    CONST robtarget T562:=[[38.419855,52.240778,11.799995],[0.000000,0.000000,1.000000,0.000000],[0,0,-1,0],[9E+09,9E+09,9E+09,9E+09,9E+09,9E+09]];
    CONST robtarget T563:=[[38.419855,76.422528,11.799995],[0.000000,0.000000,1.000000,0.000000],[0,0,-1,0],[9E+09,9E+09,9E+09,9E+09,9E+09,9E+09]];
    CONST robtarget T564:=[[38.419855,83.577479,11.799995],[0.000000,0.000000,1.000000,0.000000],[0,0,-1,0],[9E+09,9E+09,9E+09,9E+09,9E+09,9E+09]];
    CONST robtarget T565:=[[38.419855,107.759230,11.799995],[0.000000,0.000000,1.000000,0.000000],[0,0,-1,0],[9E+09,9E+09,9E+09,9E+09,9E+09,9E+09]];
    CONST robtarget T566:=[[39.679860,109.560940,11.799995],[0.000000,0.000000,1.000000,0.000000],[0,0,-1,0],[9E+09,9E+09,9E+09,9E+09,9E+09,9E+09]];
    CONST robtarget T567:=[[39.679860,85.271589,11.799995],[0.000000,0.000000,1.000000,0.000000],[0,0,-1,0],[9E+09,9E+09,9E+09,9E+09,9E+09,9E+09]];
    CONST robtarget T568:=[[39.679860,74.728418,11.799995],[0.000000,0.000000,1.000000,0.000000],[0,0,-1,0],[9E+09,9E+09,9E+09,9E+09,9E+09,9E+09]];
    CONST robtarget T569:=[[39.679860,50.439068,11.799995],[0.000000,0.000000,1.000000,0.000000],[0,0,-1,0],[9E+09,9E+09,9E+09,9E+09,9E+09,9E+09]];
    CONST robtarget T570:=[[40.939864,48.787854,11.799995],[0.000000,0.000000,1.000000,0.000000],[0,0,-1,0],[9E+09,9E+09,9E+09,9E+09,9E+09,9E+09]];
    CONST robtarget T571:=[[40.939864,73.708792,11.799995],[0.000000,0.000000,1.000000,0.000000],[0,0,-1,0],[9E+09,9E+09,9E+09,9E+09,9E+09,9E+09]];
    CONST robtarget T572:=[[40.939864,86.291215,11.799995],[0.000000,0.000000,1.000000,0.000000],[0,0,-1,0],[9E+09,9E+09,9E+09,9E+09,9E+09,9E+09]];
    CONST robtarget T573:=[[40.939864,111.212154,11.799995],[0.000000,0.000000,1.000000,0.000000],[0,0,-1,0],[9E+09,9E+09,9E+09,9E+09,9E+09,9E+09]];
    CONST robtarget T574:=[[42.199869,112.721391,11.799995],[0.000000,0.000000,1.000000,0.000000],[0,0,-1,0],[9E+09,9E+09,9E+09,9E+09,9E+09,9E+09]];
    CONST robtarget T575:=[[42.199869,86.948670,11.799995],[0.000000,0.000000,1.000000,0.000000],[0,0,-1,0],[9E+09,9E+09,9E+09,9E+09,9E+09,9E+09]];
    CONST robtarget T576:=[[42.199869,73.051337,11.799995],[0.000000,0.000000,1.000000,0.000000],[0,0,-1,0],[9E+09,9E+09,9E+09,9E+09,9E+09,9E+09]];
    CONST robtarget T577:=[[42.199869,47.278617,11.799995],[0.000000,0.000000,1.000000,0.000000],[0,0,-1,0],[9E+09,9E+09,9E+09,9E+09,9E+09,9E+09]];
    CONST robtarget T578:=[[43.459873,45.884908,11.799995],[0.000000,0.000000,1.000000,0.000000],[0,0,-1,0],[9E+09,9E+09,9E+09,9E+09,9E+09,9E+09]];
    CONST robtarget T579:=[[43.459873,72.670297,11.799995],[0.000000,0.000000,1.000000,0.000000],[0,0,-1,0],[9E+09,9E+09,9E+09,9E+09,9E+09,9E+09]];
    CONST robtarget T580:=[[43.459873,87.329711,11.799995],[0.000000,0.000000,1.000000,0.000000],[0,0,-1,0],[9E+09,9E+09,9E+09,9E+09,9E+09,9E+09]];
    CONST robtarget T581:=[[43.459873,114.115099,11.799995],[0.000000,0.000000,1.000000,0.000000],[0,0,-1,0],[9E+09,9E+09,9E+09,9E+09,9E+09,9E+09]];
    CONST robtarget T582:=[[44.719878,115.412758,11.799995],[0.000000,0.000000,1.000000,0.000000],[0,0,-1,0],[9E+09,9E+09,9E+09,9E+09,9E+09,9E+09]];
    CONST robtarget T583:=[[44.719878,87.487316,11.799995],[0.000000,0.000000,1.000000,0.000000],[0,0,-1,0],[9E+09,9E+09,9E+09,9E+09,9E+09,9E+09]];
    CONST robtarget T584:=[[44.719878,72.512692,11.799995],[0.000000,0.000000,1.000000,0.000000],[0,0,-1,0],[9E+09,9E+09,9E+09,9E+09,9E+09,9E+09]];
    CONST robtarget T585:=[[44.719878,44.587250,11.799995],[0.000000,0.000000,1.000000,0.000000],[0,0,-1,0],[9E+09,9E+09,9E+09,9E+09,9E+09,9E+09]];
    CONST robtarget T586:=[[45.979882,43.373063,11.799995],[0.000000,0.000000,1.000000,0.000000],[0,0,-1,0],[9E+09,9E+09,9E+09,9E+09,9E+09,9E+09]];
    CONST robtarget T587:=[[45.979882,72.576253,11.799995],[0.000000,0.000000,1.000000,0.000000],[0,0,-1,0],[9E+09,9E+09,9E+09,9E+09,9E+09,9E+09]];
    CONST robtarget T588:=[[45.979882,87.423755,11.799995],[0.000000,0.000000,1.000000,0.000000],[0,0,-1,0],[9E+09,9E+09,9E+09,9E+09,9E+09,9E+09]];
    CONST robtarget T589:=[[45.979882,116.626944,11.799995],[0.000000,0.000000,1.000000,0.000000],[0,0,-1,0],[9E+09,9E+09,9E+09,9E+09,9E+09,9E+09]];
    CONST robtarget T590:=[[47.239887,117.767805,11.799995],[0.000000,0.000000,1.000000,0.000000],[0,0,-1,0],[9E+09,9E+09,9E+09,9E+09,9E+09,9E+09]];
    CONST robtarget T591:=[[47.239887,87.152583,11.799995],[0.000000,0.000000,1.000000,0.000000],[0,0,-1,0],[9E+09,9E+09,9E+09,9E+09,9E+09,9E+09]];
    CONST robtarget T592:=[[47.239887,72.847425,11.799995],[0.000000,0.000000,1.000000,0.000000],[0,0,-1,0],[9E+09,9E+09,9E+09,9E+09,9E+09,9E+09]];
    CONST robtarget T593:=[[47.239887,42.232203,11.799995],[0.000000,0.000000,1.000000,0.000000],[0,0,-1,0],[9E+09,9E+09,9E+09,9E+09,9E+09,9E+09]];
    CONST robtarget T594:=[[48.499891,41.180273,11.799995],[0.000000,0.000000,1.000000,0.000000],[0,0,-1,0],[9E+09,9E+09,9E+09,9E+09,9E+09,9E+09]];
    CONST robtarget T595:=[[48.499891,73.379202,11.799995],[0.000000,0.000000,1.000000,0.000000],[0,0,-1,0],[9E+09,9E+09,9E+09,9E+09,9E+09,9E+09]];
    CONST robtarget T596:=[[48.499891,86.620805,11.799995],[0.000000,0.000000,1.000000,0.000000],[0,0,-1,0],[9E+09,9E+09,9E+09,9E+09,9E+09,9E+09]];
    CONST robtarget T597:=[[48.499891,118.819735,11.799995],[0.000000,0.000000,1.000000,0.000000],[0,0,-1,0],[9E+09,9E+09,9E+09,9E+09,9E+09,9E+09]];
    CONST robtarget T598:=[[49.759896,119.803025,11.799995],[0.000000,0.000000,1.000000,0.000000],[0,0,-1,0],[9E+09,9E+09,9E+09,9E+09,9E+09,9E+09]];
    CONST robtarget T599:=[[49.759896,85.779969,11.799995],[0.000000,0.000000,1.000000,0.000000],[0,0,-1,0],[9E+09,9E+09,9E+09,9E+09,9E+09,9E+09]];
    CONST robtarget T600:=[[49.759896,74.220038,11.799995],[0.000000,0.000000,1.000000,0.000000],[0,0,-1,0],[9E+09,9E+09,9E+09,9E+09,9E+09,9E+09]];
    CONST robtarget T601:=[[49.759896,40.196983,11.799995],[0.000000,0.000000,1.000000,0.000000],[0,0,-1,0],[9E+09,9E+09,9E+09,9E+09,9E+09,9E+09]];
    CONST robtarget T602:=[[51.019900,39.265681,11.799995],[0.000000,0.000000,1.000000,0.000000],[0,0,-1,0],[9E+09,9E+09,9E+09,9E+09,9E+09,9E+09]];
    CONST robtarget T603:=[[51.019900,75.547902,11.799995],[0.000000,0.000000,1.000000,0.000000],[0,0,-1,0],[9E+09,9E+09,9E+09,9E+09,9E+09,9E+09]];
    CONST robtarget T604:=[[51.019900,84.452106,11.799995],[0.000000,0.000000,1.000000,0.000000],[0,0,-1,0],[9E+09,9E+09,9E+09,9E+09,9E+09,9E+09]];
    CONST robtarget T605:=[[51.019900,120.734326,11.799995],[0.000000,0.000000,1.000000,0.000000],[0,0,-1,0],[9E+09,9E+09,9E+09,9E+09,9E+09,9E+09]];
    CONST robtarget T606:=[[52.279905,121.607260,11.799995],[0.000000,0.000000,1.000000,0.000000],[0,0,-1,0],[9E+09,9E+09,9E+09,9E+09,9E+09,9E+09]];
    CONST robtarget T607:=[[52.279905,81.789524,11.799995],[0.000000,0.000000,1.000000,0.000000],[0,0,-1,0],[9E+09,9E+09,9E+09,9E+09,9E+09,9E+09]];
    CONST robtarget T608:=[[52.279905,78.210483,11.799995],[0.000000,0.000000,1.000000,0.000000],[0,0,-1,0],[9E+09,9E+09,9E+09,9E+09,9E+09,9E+09]];
    CONST robtarget T609:=[[52.279905,38.392748,11.799995],[0.000000,0.000000,1.000000,0.000000],[0,0,-1,0],[9E+09,9E+09,9E+09,9E+09,9E+09,9E+09]];
    CONST robtarget T610:=[[53.539909,37.589739,11.799995],[0.000000,0.000000,1.000000,0.000000],[0,0,-1,0],[9E+09,9E+09,9E+09,9E+09,9E+09,9E+09]];
    CONST robtarget T611:=[[53.539909,122.410268,11.799995],[0.000000,0.000000,1.000000,0.000000],[0,0,-1,0],[9E+09,9E+09,9E+09,9E+09,9E+09,9E+09]];
    CONST robtarget T612:=[[54.799914,123.174878,11.799995],[0.000000,0.000000,1.000000,0.000000],[0,0,-1,0],[9E+09,9E+09,9E+09,9E+09,9E+09,9E+09]];
    CONST robtarget T613:=[[54.799914,36.825129,11.799995],[0.000000,0.000000,1.000000,0.000000],[0,0,-1,0],[9E+09,9E+09,9E+09,9E+09,9E+09,9E+09]];
    CONST robtarget T614:=[[56.059918,36.110177,11.799995],[0.000000,0.000000,1.000000,0.000000],[0,0,-1,0],[9E+09,9E+09,9E+09,9E+09,9E+09,9E+09]];
    CONST robtarget T615:=[[56.059918,123.889831,11.799995],[0.000000,0.000000,1.000000,0.000000],[0,0,-1,0],[9E+09,9E+09,9E+09,9E+09,9E+09,9E+09]];
    CONST robtarget T616:=[[57.319923,124.546114,11.799995],[0.000000,0.000000,1.000000,0.000000],[0,0,-1,0],[9E+09,9E+09,9E+09,9E+09,9E+09,9E+09]];
    CONST robtarget T617:=[[57.319923,35.453894,11.799995],[0.000000,0.000000,1.000000,0.000000],[0,0,-1,0],[9E+09,9E+09,9E+09,9E+09,9E+09,9E+09]];
    CONST robtarget T618:=[[58.579927,34.827050,11.799995],[0.000000,0.000000,1.000000,0.000000],[0,0,-1,0],[9E+09,9E+09,9E+09,9E+09,9E+09,9E+09]];
    CONST robtarget T619:=[[58.579927,125.172958,11.799995],[0.000000,0.000000,1.000000,0.000000],[0,0,-1,0],[9E+09,9E+09,9E+09,9E+09,9E+09,9E+09]];
    CONST robtarget T620:=[[59.839932,125.745278,11.799995],[0.000000,0.000000,1.000000,0.000000],[0,0,-1,0],[9E+09,9E+09,9E+09,9E+09,9E+09,9E+09]];
    CONST robtarget T621:=[[59.839932,34.254730,11.799995],[0.000000,0.000000,1.000000,0.000000],[0,0,-1,0],[9E+09,9E+09,9E+09,9E+09,9E+09,9E+09]];
    CONST robtarget T622:=[[61.099936,33.722290,11.799995],[0.000000,0.000000,1.000000,0.000000],[0,0,-1,0],[9E+09,9E+09,9E+09,9E+09,9E+09,9E+09]];
    CONST robtarget T623:=[[61.099936,126.277717,11.799995],[0.000000,0.000000,1.000000,0.000000],[0,0,-1,0],[9E+09,9E+09,9E+09,9E+09,9E+09,9E+09]];
    CONST robtarget T624:=[[62.359941,126.783143,11.799995],[0.000000,0.000000,1.000000,0.000000],[0,0,-1,0],[9E+09,9E+09,9E+09,9E+09,9E+09,9E+09]];
    CONST robtarget T625:=[[62.359941,33.216864,11.799995],[0.000000,0.000000,1.000000,0.000000],[0,0,-1,0],[9E+09,9E+09,9E+09,9E+09,9E+09,9E+09]];
    CONST robtarget T626:=[[63.619945,32.772318,11.799995],[0.000000,0.000000,1.000000,0.000000],[0,0,-1,0],[9E+09,9E+09,9E+09,9E+09,9E+09,9E+09]];
    CONST robtarget T627:=[[63.619945,127.227690,11.799995],[0.000000,0.000000,1.000000,0.000000],[0,0,-1,0],[9E+09,9E+09,9E+09,9E+09,9E+09,9E+09]];
    CONST robtarget T628:=[[64.879950,127.652167,11.799995],[0.000000,0.000000,1.000000,0.000000],[0,0,-1,0],[9E+09,9E+09,9E+09,9E+09,9E+09,9E+09]];
    CONST robtarget T629:=[[64.879950,32.347841,11.799995],[0.000000,0.000000,1.000000,0.000000],[0,0,-1,0],[9E+09,9E+09,9E+09,9E+09,9E+09,9E+09]];
    CONST robtarget T630:=[[66.139954,31.969479,11.799995],[0.000000,0.000000,1.000000,0.000000],[0,0,-1,0],[9E+09,9E+09,9E+09,9E+09,9E+09,9E+09]];
    CONST robtarget T631:=[[66.139954,128.030529,11.799995],[0.000000,0.000000,1.000000,0.000000],[0,0,-1,0],[9E+09,9E+09,9E+09,9E+09,9E+09,9E+09]];
    CONST robtarget T632:=[[67.399959,128.374988,11.799995],[0.000000,0.000000,1.000000,0.000000],[0,0,-1,0],[9E+09,9E+09,9E+09,9E+09,9E+09,9E+09]];
    CONST robtarget T633:=[[67.399959,31.625019,11.799995],[0.000000,0.000000,1.000000,0.000000],[0,0,-1,0],[9E+09,9E+09,9E+09,9E+09,9E+09,9E+09]];
    CONST robtarget T634:=[[68.659963,31.307526,11.799995],[0.000000,0.000000,1.000000,0.000000],[0,0,-1,0],[9E+09,9E+09,9E+09,9E+09,9E+09,9E+09]];
    CONST robtarget T635:=[[68.659963,128.692481,11.799995],[0.000000,0.000000,1.000000,0.000000],[0,0,-1,0],[9E+09,9E+09,9E+09,9E+09,9E+09,9E+09]];
    CONST robtarget T636:=[[69.919968,128.960575,11.799995],[0.000000,0.000000,1.000000,0.000000],[0,0,-1,0],[9E+09,9E+09,9E+09,9E+09,9E+09,9E+09]];
    CONST robtarget T637:=[[69.919968,31.039433,11.799995],[0.000000,0.000000,1.000000,0.000000],[0,0,-1,0],[9E+09,9E+09,9E+09,9E+09,9E+09,9E+09]];
    CONST robtarget T638:=[[71.179972,30.786444,11.799995],[0.000000,0.000000,1.000000,0.000000],[0,0,-1,0],[9E+09,9E+09,9E+09,9E+09,9E+09,9E+09]];
    CONST robtarget T639:=[[71.179972,129.213563,11.799995],[0.000000,0.000000,1.000000,0.000000],[0,0,-1,0],[9E+09,9E+09,9E+09,9E+09,9E+09,9E+09]];
    CONST robtarget T640:=[[72.439977,129.413129,11.799995],[0.000000,0.000000,1.000000,0.000000],[0,0,-1,0],[9E+09,9E+09,9E+09,9E+09,9E+09,9E+09]];
    CONST robtarget T641:=[[72.439977,30.586879,11.799995],[0.000000,0.000000,1.000000,0.000000],[0,0,-1,0],[9E+09,9E+09,9E+09,9E+09,9E+09,9E+09]];
    CONST robtarget T642:=[[73.699981,30.406130,11.799995],[0.000000,0.000000,1.000000,0.000000],[0,0,-1,0],[9E+09,9E+09,9E+09,9E+09,9E+09,9E+09]];
    CONST robtarget T643:=[[73.699981,40.937335,11.799995],[0.000000,0.000000,1.000000,0.000000],[0,0,-1,0],[9E+09,9E+09,9E+09,9E+09,9E+09,9E+09]];
    CONST robtarget T644:=[[73.699981,49.062665,11.799995],[0.000000,0.000000,1.000000,0.000000],[0,0,-1,0],[9E+09,9E+09,9E+09,9E+09,9E+09,9E+09]];
    CONST robtarget T645:=[[73.699981,75.937339,11.799995],[0.000000,0.000000,1.000000,0.000000],[0,0,-1,0],[9E+09,9E+09,9E+09,9E+09,9E+09,9E+09]];
    CONST robtarget T646:=[[73.699981,84.062668,11.799995],[0.000000,0.000000,1.000000,0.000000],[0,0,-1,0],[9E+09,9E+09,9E+09,9E+09,9E+09,9E+09]];
    CONST robtarget T647:=[[73.699981,110.937342,11.799995],[0.000000,0.000000,1.000000,0.000000],[0,0,-1,0],[9E+09,9E+09,9E+09,9E+09,9E+09,9E+09]];
    CONST robtarget T648:=[[73.699981,119.062672,11.799995],[0.000000,0.000000,1.000000,0.000000],[0,0,-1,0],[9E+09,9E+09,9E+09,9E+09,9E+09,9E+09]];
    CONST robtarget T649:=[[73.699981,129.593877,11.799995],[0.000000,0.000000,1.000000,0.000000],[0,0,-1,0],[9E+09,9E+09,9E+09,9E+09,9E+09,9E+09]];
    CONST robtarget T650:=[[74.959986,129.735844,11.799995],[0.000000,0.000000,1.000000,0.000000],[0,0,-1,0],[9E+09,9E+09,9E+09,9E+09,9E+09,9E+09]];
    CONST robtarget T651:=[[74.959986,120.544921,11.799995],[0.000000,0.000000,1.000000,0.000000],[0,0,-1,0],[9E+09,9E+09,9E+09,9E+09,9E+09,9E+09]];
    CONST robtarget T652:=[[74.959986,109.455091,11.799995],[0.000000,0.000000,1.000000,0.000000],[0,0,-1,0],[9E+09,9E+09,9E+09,9E+09,9E+09,9E+09]];
    CONST robtarget T653:=[[74.959986,85.544918,11.799995],[0.000000,0.000000,1.000000,0.000000],[0,0,-1,0],[9E+09,9E+09,9E+09,9E+09,9E+09,9E+09]];
    CONST robtarget T654:=[[74.959986,74.455090,11.799995],[0.000000,0.000000,1.000000,0.000000],[0,0,-1,0],[9E+09,9E+09,9E+09,9E+09,9E+09,9E+09]];
    CONST robtarget T655:=[[74.959986,50.544916,11.799995],[0.000000,0.000000,1.000000,0.000000],[0,0,-1,0],[9E+09,9E+09,9E+09,9E+09,9E+09,9E+09]];
    CONST robtarget T656:=[[74.959986,39.455086,11.799995],[0.000000,0.000000,1.000000,0.000000],[0,0,-1,0],[9E+09,9E+09,9E+09,9E+09,9E+09,9E+09]];
    CONST robtarget T657:=[[74.959986,30.264163,11.799995],[0.000000,0.000000,1.000000,0.000000],[0,0,-1,0],[9E+09,9E+09,9E+09,9E+09,9E+09,9E+09]];
    CONST robtarget T658:=[[76.219990,30.153959,11.799995],[0.000000,0.000000,1.000000,0.000000],[0,0,-1,0],[9E+09,9E+09,9E+09,9E+09,9E+09,9E+09]];
    CONST robtarget T659:=[[76.219990,38.524551,11.799995],[0.000000,0.000000,1.000000,0.000000],[0,0,-1,0],[9E+09,9E+09,9E+09,9E+09,9E+09,9E+09]];
    CONST robtarget T660:=[[76.219990,51.475451,11.799995],[0.000000,0.000000,1.000000,0.000000],[0,0,-1,0],[9E+09,9E+09,9E+09,9E+09,9E+09,9E+09]];
    CONST robtarget T661:=[[76.219990,73.524553,11.799995],[0.000000,0.000000,1.000000,0.000000],[0,0,-1,0],[9E+09,9E+09,9E+09,9E+09,9E+09,9E+09]];
    CONST robtarget T662:=[[76.219990,86.475455,11.799995],[0.000000,0.000000,1.000000,0.000000],[0,0,-1,0],[9E+09,9E+09,9E+09,9E+09,9E+09,9E+09]];
    CONST robtarget T663:=[[76.219990,108.524556,11.799995],[0.000000,0.000000,1.000000,0.000000],[0,0,-1,0],[9E+09,9E+09,9E+09,9E+09,9E+09,9E+09]];
    CONST robtarget T664:=[[76.219990,121.475457,11.799995],[0.000000,0.000000,1.000000,0.000000],[0,0,-1,0],[9E+09,9E+09,9E+09,9E+09,9E+09,9E+09]];
    CONST robtarget T665:=[[76.219990,129.846049,11.799995],[0.000000,0.000000,1.000000,0.000000],[0,0,-1,0],[9E+09,9E+09,9E+09,9E+09,9E+09,9E+09]];
    CONST robtarget T666:=[[77.479995,129.931001,11.799995],[0.000000,0.000000,1.000000,0.000000],[0,0,-1,0],[9E+09,9E+09,9E+09,9E+09,9E+09,9E+09]];
    CONST robtarget T667:=[[77.479995,122.050628,11.799995],[0.000000,0.000000,1.000000,0.000000],[0,0,-1,0],[9E+09,9E+09,9E+09,9E+09,9E+09,9E+09]];
    CONST robtarget T668:=[[77.479995,107.949384,11.799995],[0.000000,0.000000,1.000000,0.000000],[0,0,-1,0],[9E+09,9E+09,9E+09,9E+09,9E+09,9E+09]];
